# B&R Automation Studio project TD52 (part 145)

#### ECB_Test.st - Implementation code
```iecst
(********************************************************************
 * COPYRIGHT -- INNIO Company
 ********************************************************************
 * Program: ECB_Test
 * File: ECB_Test.st
 * Author: 502423184
 * Created: January 12, 2018
 ********************************************************************
 * Implementation of program ECB_Test
 ********************************************************************)

PROGRAM _INIT

	(** INIT: Disable PBC_Buffer Task *)
	bECB_Buffer_Test	:=	TRUE;

	(** Bit Names **)
	Buffer.Bits[0].used	:=	8;
	Buffer.Bits[1].used	:=	0;
	Buffer.Bits[0].Info[0].Name			:=	'GCB_ON';
	Buffer.Bits[0].Info[1].Name			:=	'Trip_1';
	Buffer.Bits[0].Info[2].Name			:=	'Trip_2';
	Buffer.Bits[0].Info[3].Name			:=	'Trip_3';
	Buffer.Bits[0].Info[4].Name			:=	'GrC_VoltageLow';
	Buffer.Bits[0].Info[5].Name			:=	'GrC_SpeedChange';
	Buffer.Bits[0].Info[6].Name			:=	'GrC_CurrentChange';
	Buffer.Bits[0].Info[7].Name			:=	'FS_IPOffs_Trip';
	Buffer.Bits[1].Info[0].Name			:=	'';
	Buffer.Bits[1].Info[1].Name			:=	'';
	Buffer.Bits[1].Info[2].Name			:=	'';
	Buffer.Bits[1].Info[3].Name			:=	'';

	(** Bit Pattern Names **)
	Buffer.pattern[0].Name		:=	 'PBCNegVoltCheck_';
	Buffer.pattern[1].Name		:=	 'PBCNegPresCheck_';
	Buffer.pattern[2].Name		:=	 'PBCPresSlopeCheck_';
	Buffer.pattern[3].Name		:=	 'PBCSlowDriftCheck_';
	Buffer.pattern[4].Name		:=	 'PBCMemBurst_';
	Buffer.pattern[5].Name		:=	 'PBCSensError_';
	Buffer.pattern[6].Name		:=	 'GlowIgn_';
	Buffer.pattern[7].Name		:=	 'Misfire_I_';
	Buffer.pattern[8].Name		:=	 'Misfire_II_';
	Buffer.pattern[9].Name		:=	 'SkipFire_';
	Buffer.pattern[10].Name		:=	 'LimpHome_';
	Buffer.pattern[11].Name		:=	 'LimpHomeExt_';
	Buffer.pattern[12].Name		:=	 '';
	Buffer.pattern[13].Name		:=	 '';
	Buffer.pattern[14].Name		:=	 '';
	Buffer.pattern[15].Name		:=	 '';
	Buffer.pattern[16].Name		:=	 '';

	Buffer.iCnt_pattern			:=	15;

	(** ui16 Names, Conversions, Signs and Units *)
	iCnt	:=	0;
	FOR iSet:=0 TO 304 BY 16 DO
		Buffer.ui16[iSet].Name 	:=	'Ign_Timing_';		Buffer.ui16[iSet].Co := 100;	Buffer.ui16[iSet].Signed := 1;	Buffer.ui16[iSet].Unit := '°CA';
		iCnt := iCnt +1;	itoa(iCnt,ADR(strCnt));		strcat(ADR(Buffer.ui16[iSet].Name), ADR(strCnt));
	END_FOR
	iCnt	:=	0;
	FOR iSet:=1 TO 305 BY 16 DO
		Buffer.ui16[iSet].Name := 'Knck_Intgr_';		Buffer.ui16[iSet].Co := 10;		Buffer.ui16[iSet].Signed := 1;	Buffer.ui16[iSet].Unit := '%';
		iCnt := iCnt +1;	itoa(iCnt,ADR(strCnt));		strcat(ADR(Buffer.ui16[iSet].Name), ADR(strCnt));
	END_FOR
	iCnt	:=	0;
	FOR iSet:=2 TO 306 BY 16 DO
		Buffer.ui16[iSet].Name := 'U_Ign_';				Buffer.ui16[iSet].Co := 1;		Buffer.ui16[iSet].Signed := 0;	Buffer.ui16[iSet].Unit := 'kV';
		iCnt := iCnt +1;	itoa(iCnt,ADR(strCnt));		strcat(ADR(Buffer.ui16[iSet].Name), ADR(strCnt));
	END_FOR
	iCnt	:=	0;
	FOR iSet:=3 TO 307 BY 16 DO
		Buffer.ui16[iSet].Name := 'PI_Duration_';		Buffer.ui16[iSet].Co := 100;	Buffer.ui16[iSet].Signed := 0;	Buffer.ui16[iSet].Unit := '°CA';
		iCnt := iCnt +1;	itoa(iCnt,ADR(strCnt));		strcat(ADR(Buffer.ui16[iSet].Name), ADR(strCnt));
	END_FOR
	iCnt	:=	0;
	FOR iSet:=4 TO 308 BY 16 DO
		Buffer.ui16[iSet].Name := 'PI_Dur_Map_Offs_';	Buffer.ui16[iSet].Co := 1000;	Buffer.ui16[iSet].Signed := 1;	Buffer.ui16[iSet].Unit := '%';
		iCnt := iCnt +1;	itoa(iCnt,ADR(strCnt));		strcat(ADR(Buffer.ui16[iSet].Name), ADR(strCnt));
	END_FOR
	iCnt	:=	0;
	FOR iSet:=6 TO 310 BY 16 DO
		Buffer.ui16[iSet].Name := 'Pr_Knock_';			Buffer.ui16[iSet].Co := 100;	Buffer.ui16[iSet].Signed := 0;	Buffer.ui16[iSet].Unit := 'bar';
		iCnt := iCnt +1;	itoa(iCnt,ADR(strCnt));		strcat(ADR(Buffer.ui16[iSet].Name), ADR(strCnt));
	END_FOR
	iCnt	:=	0;
	FOR iSet:=7 TO 311 BY 16 DO
		Buffer.ui16[iSet].Name := 'Pr_Knock_Filt_';		Buffer.ui16[iSet].Co := 100;	Buffer.ui16[iSet].Signed := 0;	Buffer.ui16[iSet].Unit := 'bar';
		iCnt := iCnt +1;	itoa(iCnt,ADR(strCnt));		strcat(ADR(Buffer.ui16[iSet].Name), ADR(strCnt));
	END_FOR
	iCnt	:=	0;
	FOR iSet:=8 TO 312 BY 16 DO
		Buffer.ui16[iSet].Name := 'Pr_Peak_';			Buffer.ui16[iSet].Co := 100;	Buffer.ui16[iSet].Signed := 0;	Buffer.ui16[iSet].Unit := 'bar';
		iCnt := iCnt +1;	itoa(iCnt,ADR(strCnt));		strcat(ADR(Buffer.ui16[iSet].Name), ADR(strCnt));
	END_FOR
	iCnt	:=	0;
	FOR iSet:=9 TO 313 BY 16 DO
		Buffer.ui16[iSet].Name := 'Pr_Peak_Filt_';		Buffer.ui16[iSet].Co := 100;	Buffer.ui16[iSet].Signed := 0;	Buffer.ui16[iSet].Unit := 'bar';
		iCnt := iCnt +1;	itoa(iCnt,ADR(strCnt));		strcat(ADR(Buffer.ui16[iSet].Name), ADR(strCnt));
	END_FOR
	iCnt	:=	0;
	FOR iSet:=10 TO 314 BY 16 DO
		Buffer.ui16[iSet].Name := 'Pr_IMEP_';			Buffer.ui16[iSet].Co := 100;	Buffer.ui16[iSet].Signed := 0;	Buffer.ui16[iSet].Unit := 'bar';
		iCnt := iCnt +1;	itoa(iCnt,ADR(strCnt));		strcat(ADR(Buffer.ui16[iSet].Name), ADR(strCnt));
	END_FOR
	iCnt	:=	0;
	FOR iSet:=11 TO 315 BY 16 DO
		Buffer.ui16[iSet].Name := 'Pr_49bfTDC_';		Buffer.ui16[iSet].Co := 100;	Buffer.ui16[iSet].Signed := 0;	Buffer.ui16[iSet].Unit := 'bar';
		iCnt := iCnt +1;	itoa(iCnt,ADR(strCnt));		strcat(ADR(Buffer.ui16[iSet].Name), ADR(strCnt));
	END_FOR
	iCnt	:=	0;
	FOR iSet:=12 TO 316 BY 16 DO
		Buffer.ui16[iSet].Name := 'Pr_49afTDC_';		Buffer.ui16[iSet].Co := 100;	Buffer.ui16[iSet].Signed := 0;	Buffer.ui16[iSet].Unit := 'bar';
		iCnt := iCnt +1;	itoa(iCnt,ADR(strCnt));		strcat(ADR(Buffer.ui16[iSet].Name), ADR(strCnt));
	END_FOR
	iCnt	:=	0;
	FOR iSet:=13 TO 317 BY 16 DO
		Buffer.ui16[iSet].Name := 'MFBvar_';			Buffer.ui16[iSet].Co := 100;	Buffer.ui16[iSet].Signed := 1;	Buffer.ui16[iSet].Unit := '°CA';
		iCnt := iCnt +1;	itoa(iCnt,ADR(strCnt));		strcat(ADR(Buffer.ui16[iSet].Name), ADR(strCnt));
	END_FOR
	iCnt	:=	0;
	FOR iSet:=14 TO 318 BY 16 DO
		Buffer.ui16[iSet].Name := 'Pr_Knock_Lim_';		Buffer.ui16[iSet].Co := 100;	Buffer.ui16[iSet].Signed := 0;	Buffer.ui16[iSet].Unit := 'bar';
		iCnt := iCnt +1;	itoa(iCnt,ADR(strCnt));		strcat(ADR(Buffer.ui16[iSet].Name), ADR(strCnt));
	END_FOR

	Buffer.iCnt_ui16			:=	326;

	(** ui16_H Names, Conversions, Signs and Units *)
	Buffer.ui16_H[0].Name := 'N_Eng';			Buffer.ui16_H[0].Co := 10;		Buffer.ui16_H[0].Signed := 0;	Buffer.ui16_H[0].Unit := 'rpm';
	Buffer.ui16_H[1].Name := 'P_Set';			Buffer.ui16_H[1].Co	:= 1;		Buffer.ui16_H[1].Signed := 0;	Buffer.ui16_H[1].Unit := 'kW';
	Buffer.ui16_H[2].Name := 'P_Act';			Buffer.ui16_H[2].Co := 1;		Buffer.ui16_H[2].Signed	:= 1;	Buffer.ui16_H[2].Unit := 'kW';
	Buffer.ui16_H[3].Name := 'Q_Act';			Buffer.ui16_H[3].Co := 1;		Buffer.ui16_H[3].Signed	:= 1;	Buffer.ui16_H[3].Unit := 'kVAr';
	Buffer.ui16_H[4].Name := 'U_L1L2';			Buffer.ui16_H[4].Co := 1;		Buffer.ui16_H[4].Signed	:= 1;	Buffer.ui16_H[4].Unit := 'V';
	Buffer.ui16_H[5].Name := 'U_L2L3';			Buffer.ui16_H[5].Co := 1;		Buffer.ui16_H[5].Signed	:= 1;	Buffer.ui16_H[5].Unit := 'V';
	Buffer.ui16_H[6].Name := 'U_L3L1';			Buffer.ui16_H[6].Co := 1;		Buffer.ui16_H[6].Signed	:= 1;	Buffer.ui16_H[6].Unit := 'V';
	Buffer.ui16_H[7].Name := 'I_L1';			Buffer.ui16_H[7].Co := 1;		Buffer.ui16_H[7].Signed	:= 1;	Buffer.ui16_H[7].Unit := 'A';
	Buffer.ui16_H[8].Name := 'I_L2';			Buffer.ui16_H[8].Co := 1;		Buffer.ui16_H[8].Signed	:= 1;	Buffer.ui16_H[8].Unit := 'A';
	Buffer.ui16_H[9].Name := 'I_L3';			Buffer.ui16_H[9].Co := 1;		Buffer.ui16_H[9].Signed	:= 1;	Buffer.ui16_H[9].Unit := 'A';
	Buffer.ui16_H[10].Name := 'Frequency';		Buffer.ui16_H[10].Co := 1000;	Buffer.ui16_H[10].Signed := 0;	Buffer.ui16_H[10].Unit := 'Hz';
	Buffer.ui16_H[11].Name := 'CosPhi';			Buffer.ui16_H[11].Co := 100;	Buffer.ui16_H[11].Signed := 1;	Buffer.ui16_H[11].Unit := '';
	Buffer.ui16_H[12].Name := 'Lambda_Set';		Buffer.ui16_H[12].Co := 1000;	Buffer.ui16_H[12].Signed := 0;	Buffer.ui16_H[12].Unit := '';
	Buffer.ui16_H[13].Name := 'Pr_Leanox_Set';	Buffer.ui16_H[13].Co := 1000;	Buffer.ui16_H[13].Signed := 0;	Buffer.ui16_H[13].Unit := '';
	Buffer.ui16_H[14].Name := 'N_TCHP_A';		Buffer.ui16_H[14].Co := 0.1;	Buffer.ui16_H[14].Signed := 0;	Buffer.ui16_H[14].Unit := 'rpm';
	Buffer.ui16_H[15].Name := 'N_TCHP_B';		Buffer.ui16_H[15].Co := 0.1;	Buffer.ui16_H[15].Signed := 0;	Buffer.ui16_H[15].Unit := 'rpm';
	Buffer.ui16_H[16].Name := 'N_TCLP_A';		Buffer.ui16_H[16].Co := 0.1;	Buffer.ui16_H[16].Signed := 0;	Buffer.ui16_H[16].Unit := 'rpm';
	Buffer.ui16_H[17].Name := 'N_TCLP_B';		Buffer.ui16_H[17].Co := 0.1;	Buffer.ui16_H[17].Signed := 0;	Buffer.ui16_H[17].Unit := 'rpm';
	Buffer.ui16_H[18].Name := 'Pr_GR_Act';		Buffer.ui16_H[18].Co := 1000;	Buffer.ui16_H[18].Signed := 0;	Buffer.ui16_H[18].Unit := 'bar';
	Buffer.ui16_H[19].Name := 'Pr_GR_Set';		Buffer.ui16_H[19].Co := 1000;	Buffer.ui16_H[19].Signed := 0;	Buffer.ui16_H[19].Unit := 'bar';
	Buffer.ui16_H[20].Name := 'Pr_PC_Act';		Buffer.ui16_H[20].Co := 1000;	Buffer.ui16_H[20].Signed := 0;	Buffer.ui16_H[20].Unit := 'bar';
	Buffer.ui16_H[21].Name := 'Pr_PC_Set';		Buffer.ui16_H[21].Co := 1000;	Buffer.ui16_H[21].Signed := 0;	Buffer.ui16_H[21].Unit := 'bar';
	Buffer.ui16_H[22].Name := 'Pr_Crank_Case';	Buffer.ui16_H[22].Co := 1000;	Buffer.ui16_H[22].Signed := 1;	Buffer.ui16_H[22].Unit := 'mbar';
	Buffer.ui16_H[23].Name := 'Pos_CBV_Set';	Buffer.ui16_H[23].Co := 1000;	Buffer.ui16_H[23].Signed := 0;	Buffer.ui16_H[23].Unit := '';
	Buffer.ui16_H[24].Name := 'Pos_CBV_Act_A1';	Buffer.ui16_H[24].Co := 1000;	Buffer.ui16_H[24].Signed := 0;	Buffer.ui16_H[24].Unit := '';
	Buffer.ui16_H[25].Name := 'Pos_CBV_Act_B1';	Buffer.ui16_H[25].Co := 1000;	Buffer.ui16_H[25].Signed := 0;	Buffer.ui16_H[25].Unit := '';
	Buffer.ui16_H[26].Name := 'Pos_WG_Set';		Buffer.ui16_H[26].Co := 1000;	Buffer.ui16_H[26].Signed := 0;	Buffer.ui16_H[26].Unit := '';
	Buffer.ui16_H[27].Name := 'Pos_WG_Act_A';	Buffer.ui16_H[27].Co := 1000;	Buffer.ui16_H[27].Signed := 0;	Buffer.ui16_H[27].Unit := '';
	Buffer.ui16_H[28].Name := 'Pos_WG_Act_B';	Buffer.ui16_H[28].Co := 1000;	Buffer.ui16_H[28].Signed := 0;	Buffer.ui16_H[28].Unit := '';
	Buffer.ui16_H[29].Name := 'Pr_P1HP_A';		Buffer.ui16_H[29].Co := 1000;	Buffer.ui16_H[29].Signed := 0;	Buffer.ui16_H[29].Unit := 'bar';
	Buffer.ui16_H[30].Name := 'Pr_P1HP_B';		Buffer.ui16_H[30].Co := 1000;	Buffer.ui16_H[30].Signed := 0;	Buffer.ui16_H[30].Unit := 'bar';
	Buffer.ui16_H[31].Name := 'Pr_P2s_A';		Buffer.ui16_H[31].Co := 1000;	Buffer.ui16_H[31].Signed := 0;	Buffer.ui16_H[31].Unit := 'bar';
	Buffer.ui16_H[32].Name := 'Pr_P2s_B';		Buffer.ui16_H[32].Co := 1000;	Buffer.ui16_H[32].Signed := 0;	Buffer.ui16_H[32].Unit := 'bar';
	Buffer.ui16_H[33].Name := 'Pr_P3HP_A';		Buffer.ui16_H[33].Co := 1000;	Buffer.ui16_H[33].Signed := 0;	Buffer.ui16_H[33].Unit := 'bar';
	Buffer.ui16_H[34].Name := 'Pr_P3HP_B';		Buffer.ui16_H[34].Co := 1000;	Buffer.ui16_H[34].Signed := 0;	Buffer.ui16_H[34].Unit := 'bar';
	Buffer.ui16_H[35].Name := 'Pr_P3LP_A';		Buffer.ui16_H[35].Co := 1000;	Buffer.ui16_H[35].Signed := 0;	Buffer.ui16_H[35].Unit := 'bar';
	Buffer.ui16_H[36].Name := 'Pr_P3LP_B';		Buffer.ui16_H[36].Co := 1000;	Buffer.ui16_H[36].Signed := 0;	Buffer.ui16_H[36].Unit := 'bar';
	Buffer.ui16_H[37].Name := 'Pr_P4LP_A';		Buffer.ui16_H[37].Co := 1000;	Buffer.ui16_H[37].Signed := 0;	Buffer.ui16_H[37].Unit := 'bar';
	Buffer.ui16_H[38].Name := 'Pr_P4LP_B';		Buffer.ui16_H[38].Co := 1000;	Buffer.ui16_H[38].Signed := 0;	Buffer.ui16_H[38].Unit := 'bar';
	Buffer.ui16_H[39].Name := 'Pr_ECW';			Buffer.ui16_H[39].Co := 1000;	Buffer.ui16_H[39].Signed := 0;	Buffer.ui16_H[39].Unit := 'bar';
	Buffer.ui16_H[40].Name := 'Pr_EO';			Buffer.ui16_H[40].Co := 1000;	Buffer.ui16_H[40].Signed := 0;	Buffer.ui16_H[40].Unit := 'bar';
	Buffer.ui16_H[41].Name := 'NOx_Sensor_1';	Buffer.ui16_H[41].Co := 1;		Buffer.ui16_H[41].Signed := 0;	Buffer.ui16_H[41].Unit := '';
	Buffer.ui16_H[42].Name := 'NOx_Sensor_2';	Buffer.ui16_H[42].Co := 1;		Buffer.ui16_H[42].Signed := 0;	Buffer.ui16_H[42].Unit := '';
	Buffer.ui16_H[43].Name := 'O2_Sensor_1';	Buffer.ui16_H[43].Co := 1;		Buffer.ui16_H[43].Signed := 0;	Buffer.ui16_H[43].Unit := '';
	Buffer.ui16_H[44].Name := 'O2_Sensor_2';	Buffer.ui16_H[44].Co := 1;		Buffer.ui16_H[44].Signed := 0;	Buffer.ui16_H[44].Unit := '';
	Buffer.ui16_H[45].Name := '';				Buffer.ui16_H[45].Co := 0;		Buffer.ui16_H[45].Signed := 0;	Buffer.ui16_H[45].Unit := '';
	Buffer.ui16_H[46].Name := '';				Buffer.ui16_H[46].Co := 0;		Buffer.ui16_H[46].Signed := 0;	Buffer.ui16_H[46].Unit := '';

	Buffer.iCnt_ui16_H	:=	44;

	(** ui16_L Names, Conversions, Signs and Units *)
	FOR iSet:=0 TO 56 DO
		Buffer.ui16_low[iSet].Signed	:= 0;
		Buffer.ui16_low[iSet].Unit		:= '°C';
		Buffer.ui16_low[iSet].Co		:=	100;
	END_FOR

	Buffer.ui16_low[0].Name := 'T_T2s';
	Buffer.ui16_low[1].Name := 'T_T3HP_A';		Buffer.ui16_low[1].Co := 10;	(* nur EG temps mit Conversion 10 *)
	Buffer.ui16_low[2].Name := 'T_T3HP_B';		Buffer.ui16_low[2].Co := 10;
	Buffer.ui16_low[3].Name := 'T_T3LP_A';		Buffer.ui16_low[3].Co := 10;
	Buffer.ui16_low[4].Name := 'T_T3LP_B';		Buffer.ui16_low[4].Co := 10;
	Buffer.ui16_low[5].Name := 'T_EG_LimMax';	Buffer.ui16_low[5].Co := 10;

	iCnt	:=	0; (* zyl 1 bis 11 *)
	FOR iSet:=6 TO 36 BY 3 DO
		iCnt := iCnt +1;	itoa(iCnt,ADR(strCnt));
		Buffer.ui16_low[iSet].Name		:= 'T_EG_Cyl_';		strcat(ADR(Buffer.ui16_low[iSet].Name), ADR(strCnt));
		Buffer.ui16_low[iSet+1].Name	:= 'T_CBearing_';	strcat(ADR(Buffer.ui16_low[iSet+1].Name), ADR(strCnt));
		Buffer.ui16_low[iSet+2].Name	:= 'T_MBearing_';	strcat(ADR(Buffer.ui16_low[iSet+2].Name), ADR(strCnt));
	END_FOR
	iCnt	:=	11;	(* zyl 12 bis 20 *)
	FOR iSet:=39 TO 55 BY 2 DO
		iCnt := iCnt +1;	itoa(iCnt,ADR(strCnt));
		Buffer.ui16_low[iSet].Name		:= 'T_EG_Cyl_';		strcat(ADR(Buffer.ui16_low[iSet].Name), ADR(strCnt));
		Buffer.ui16_low[iSet+1].Name	:= 'T_CBearing_';	strcat(ADR(Buffer.ui16_low[iSet+1].Name), ADR(strCnt));
	END_FOR

	Buffer.ui16_low[57].Name := '';	Buffer.ui16_low[57].Co := 0;	Buffer.ui16_low[57].Signed := 0;	Buffer.ui16_low[57].Unit := '';

	Buffer.iCnt_ui16_low		:=	56;

END_PROGRAM

PROGRAM _CYCLIC

(** 1: is PBCMem enabled? *)
IF bPBC_Mem_Ena THEN

(** 6: save data to buffer? @control *)
	IF 	bPBC_NewData AND bPBC_Record THEN

(** 6.1: save the time *)
		Buffer.timer[iCnt_Cycle]	:= tiStamp;
(* _______________________________________________________ FAKE BITS _______________________________________________________ *)

		Buffer.Bits[0].ucData[iCnt_Cycle]	:=	1;
		Buffer.Bits[1].ucData[iCnt_Cycle]	:=	0;
		FOR iSet:= 1 TO 16 DO
			Buffer.pattern[iSet].BitPattern[iCnt_Cycle]	:=	INT_TO_UDINT(iCnt_Cycle) + INT_TO_UDINT(iCnt_Cycle)*1000;
		END_FOR

(* _______________________________________________________ FAKE PATTERNS _______________________________________________________ *)

	iCnt_Cycle10	:=	LIMIT(0,iCnt_Cycle/10,100);

	iCnt := 0;	FOR iSet:=0 TO 304 BY 16 DO			Buffer.ui16[iSet].Data[iCnt_Cycle] := 1914;			END_FOR
	iCnt := 0;	FOR iSet:=1 TO 305 BY 16 DO			Buffer.ui16[iSet].Data[iCnt_Cycle] := 43;			END_FOR
	iCnt := 0;	FOR iSet:=2 TO 306 BY 16 DO			Buffer.ui16[iSet].Data[iCnt_Cycle] := 15;			END_FOR
	iCnt := 0;	FOR iSet:=3 TO 307 BY 16 DO			Buffer.ui16[iSet].Data[iCnt_Cycle] := 6210;			END_FOR
	iCnt := 0;	FOR iSet:=4 TO 308 BY 16 DO			Buffer.ui16[iSet].Data[iCnt_Cycle] := 1492;			END_FOR
(* 5 fehlt *)
	iCnt := 0;	FOR iSet:=6 TO 310 BY 16 DO			Buffer.ui16[iSet].Data[iCnt_Cycle] := 166;			END_FOR
	iCnt := 0;	FOR iSet:=7 TO 311 BY 16 DO			Buffer.ui16[iSet].Data[iCnt_Cycle] := 166;			END_FOR
	iCnt := 0;	FOR iSet:=8 TO 312 BY 16 DO			Buffer.ui16[iSet].Data[iCnt_Cycle] := 15816;		END_FOR
	iCnt := 0;	FOR iSet:=9 TO 313 BY 16 DO			Buffer.ui16[iSet].Data[iCnt_Cycle] := 15816;		END_FOR
	iCnt := 0;	FOR iSet:=10 TO 314 BY 16 DO		Buffer.ui16[iSet].Data[iCnt_Cycle] := 2611;			END_FOR
	iCnt := 0;	FOR iSet:=11 TO 315 BY 16 DO		Buffer.ui16[iSet].Data[iCnt_Cycle] := 2233;			END_FOR
	iCnt := 0;	FOR iSet:=12 TO 316 BY 16 DO		Buffer.ui16[iSet].Data[iCnt_Cycle] := 5914;			END_FOR
	iCnt := 0;	FOR iSet:=13 TO 317 BY 16 DO		Buffer.ui16[iSet].Data[iCnt_Cycle] := 1000;			END_FOR
	iCnt := 0;	FOR iSet:=14 TO 318 BY 16 DO		Buffer.ui16[iSet].Data[iCnt_Cycle] := 2233;			END_FOR
	iCnt := 0;	FOR iSet:=15 TO 319 BY 16 DO		Buffer.ui16[iSet].Data[iCnt_Cycle] := 65293;		END_FOR
	iCnt := 0;	FOR iSet:=16 TO 320 BY 16 DO		Buffer.ui16[iSet].Data[iCnt_Cycle] := 166;			END_FOR

	Buffer.ui16_H[0].Hi[iCnt_Cycle] := 10000;		Buffer.ui16_H[0].Lo[iCnt_Cycle] := 9990;
	Buffer.ui16_H[1].Hi[iCnt_Cycle] := 10380;		Buffer.ui16_H[1].Lo[iCnt_Cycle] := 10340;
	Buffer.ui16_H[2].Hi[iCnt_Cycle] := 10434;		Buffer.ui16_H[2].Lo[iCnt_Cycle] := 10428;
	Buffer.ui16_H[3].Hi[iCnt_Cycle] := 26;			Buffer.ui16_H[3].Lo[iCnt_Cycle] := 34;
	Buffer.ui16_H[4].Hi[iCnt_Cycle] := 10621;		Buffer.ui16_H[4].Lo[iCnt_Cycle] := 10622;
	Buffer.ui16_H[5].Hi[iCnt_Cycle] := 10621;		Buffer.ui16_H[5].Lo[iCnt_Cycle] := 10622;
	Buffer.ui16_H[6].Hi[iCnt_Cycle] := 10621;		Buffer.ui16_H[6].Lo[iCnt_Cycle] := 10622;
	Buffer.ui16_H[7].Hi[iCnt_Cycle] := 568;			Buffer.ui16_H[7].Lo[iCnt_Cycle] := 569;
	Buffer.ui16_H[8].Hi[iCnt_Cycle] := 568;			Buffer.ui16_H[8].Lo[iCnt_Cycle] := 568;
	Buffer.ui16_H[9].Hi[iCnt_Cycle] := 574;			Buffer.ui16_H[9].Lo[iCnt_Cycle] := 571;
	Buffer.ui16_H[10].Hi[iCnt_Cycle] := 50000;		Buffer.ui16_H[10].Lo[iCnt_Cycle] := 49990;
	Buffer.ui16_H[11].Hi[iCnt_Cycle] := 100;		Buffer.ui16_H[11].Lo[iCnt_Cycle] := 100;
	Buffer.ui16_H[12].Hi[iCnt_Cycle] := 1973;		Buffer.ui16_H[12].Lo[iCnt_Cycle] := 1973;
	Buffer.ui16_H[13].Hi[iCnt_Cycle] := 7630;		Buffer.ui16_H[13].Lo[iCnt_Cycle] := 7630;
	Buffer.ui16_H[14].Hi[iCnt_Cycle] := 2760;		Buffer.ui16_H[14].Lo[iCnt_Cycle] := 2763;
	Buffer.ui16_H[15].Hi[iCnt_Cycle] := 2753;		Buffer.ui16_H[15].Lo[iCnt_Cycle] := 2753;
	Buffer.ui16_H[16].Hi[iCnt_Cycle] := 2625;		Buffer.ui16_H[16].Lo[iCnt_Cycle] := 2596;
	Buffer.ui16_H[17].Hi[iCnt_Cycle] := 2594;		Buffer.ui16_H[17].Lo[iCnt_Cycle] := 2594;
	Buffer.ui16_H[18].Hi[iCnt_Cycle] := 8815;		Buffer.ui16_H[18].Lo[iCnt_Cycle] := 8818;
	Buffer.ui16_H[19].Hi[iCnt_Cycle] := 8853;		Buffer.ui16_H[19].Lo[iCnt_Cycle] := 8853;
	Buffer.ui16_H[20].Hi[iCnt_Cycle] := 5369;		Buffer.ui16_H[20].Lo[iCnt_Cycle] := 5369;
	Buffer.ui16_H[21].Hi[iCnt_Cycle] := 6851;		Buffer.ui16_H[21].Lo[iCnt_Cycle] := 6851;
	Buffer.ui16_H[22].Hi[iCnt_Cycle] := 62867;		Buffer.ui16_H[22].Lo[iCnt_Cycle] := 62987;
	Buffer.ui16_H[23].Hi[iCnt_Cycle] := 28;			Buffer.ui16_H[23].Lo[iCnt_Cycle] := 28;
	Buffer.ui16_H[24].Hi[iCnt_Cycle] := 29;			Buffer.ui16_H[24].Lo[iCnt_Cycle] := 28;
	Buffer.ui16_H[25].Hi[iCnt_Cycle] := 26;			Buffer.ui16_H[25].Lo[iCnt_Cycle] := 25;
	Buffer.ui16_H[26].Hi[iCnt_Cycle] := 478;		Buffer.ui16_H[26].Lo[iCnt_Cycle] := 478;
	Buffer.ui16_H[27].Hi[iCnt_Cycle] := 487;		Buffer.ui16_H[27].Lo[iCnt_Cycle] := 486;
	Buffer.ui16_H[28].Hi[iCnt_Cycle] := 488;		Buffer.ui16_H[28].Lo[iCnt_Cycle] := 488;
	Buffer.ui16_H[29].Hi[iCnt_Cycle] := 3210;		Buffer.ui16_H[29].Lo[iCnt_Cycle] := 3213;
	Buffer.ui16_H[30].Hi[iCnt_Cycle] := 3236;		Buffer.ui16_H[30].Lo[iCnt_Cycle] := 3233;
	Buffer.ui16_H[31].Hi[iCnt_Cycle] := 6732;		Buffer.ui16_H[31].Lo[iCnt_Cycle] := 6733;
	Buffer.ui16_H[32].Hi[iCnt_Cycle] := 6662;		Buffer.ui16_H[32].Lo[iCnt_Cycle] := 6662;
	Buffer.ui16_H[33].Hi[iCnt_Cycle] := 4605;		Buffer.ui16_H[33].Lo[iCnt_Cycle] := 4621;
	Buffer.ui16_H[34].Hi[iCnt_Cycle] := 4675;		Buffer.ui16_H[34].Lo[iCnt_Cycle] := 4675;
	Buffer.ui16_H[35].Hi[iCnt_Cycle] := 2864;		Buffer.ui16_H[35].Lo[iCnt_Cycle] := 2873;
	Buffer.ui16_H[36].Hi[iCnt_Cycle] := 2879;		Buffer.ui16_H[36].Lo[iCnt_Cycle] := 2870;
	Buffer.ui16_H[37].Hi[iCnt_Cycle] := 1026;		Buffer.ui16_H[37].Lo[iCnt_Cycle] := 1029;
	Buffer.ui16_H[38].Hi[iCnt_Cycle] := 1021;		Buffer.ui16_H[38].Lo[iCnt_Cycle] := 1017;
	Buffer.ui16_H[39].Hi[iCnt_Cycle] := 2147;		Buffer.ui16_H[39].Lo[iCnt_Cycle] := 2128;
	Buffer.ui16_H[40].Hi[iCnt_Cycle] := 5797;		Buffer.ui16_H[40].Lo[iCnt_Cycle] := 5794;
	Buffer.ui16_H[41].Hi[iCnt_Cycle] := 216;		Buffer.ui16_H[41].Lo[iCnt_Cycle] := 216;
	Buffer.ui16_H[42].Hi[iCnt_Cycle] := 219;		Buffer.ui16_H[42].Lo[iCnt_Cycle] := 219;
	Buffer.ui16_H[43].Hi[iCnt_Cycle] := 0;			Buffer.ui16_H[43].Lo[iCnt_Cycle] := 0;
	Buffer.ui16_H[44].Hi[iCnt_Cycle] := 0;			Buffer.ui16_H[44].Lo[iCnt_Cycle] := 0;
	Buffer.ui16_H[45].Hi[iCnt_Cycle] := 0;			Buffer.ui16_H[45].Lo[iCnt_Cycle] := 0;
	Buffer.ui16_H[46].Hi[iCnt_Cycle] := 0;			Buffer.ui16_H[46].Lo[iCnt_Cycle] := 0;

	Buffer.ui16_low[0].Data[iCnt_Cycle10] := 7545;
	Buffer.ui16_low[1].Data[iCnt_Cycle10] := 5366;
	Buffer.ui16_low[2].Data[iCnt_Cycle10] := 5366;
	Buffer.ui16_low[3].Data[iCnt_Cycle10] := 4577;
	Buffer.ui16_low[4].Data[iCnt_Cycle10] := 4605;
	Buffer.ui16_low[5].Data[iCnt_Cycle10] := 6000;

	FOR iSet:=6 TO 36 BY 3 DO
		Buffer.ui16_low[iSet].Data[iCnt_Cycle10]	:= 52900;		(* 6,9,12 bis 36 *)
		Buffer.ui16_low[iSet+1].Data[iCnt_Cycle10]	:= 10100;		(* 7,10,13 bis 37 *)
		Buffer.ui16_low[iSet+2].Data[iCnt_Cycle10]	:= 10120;		(* 8,11,14 bis 38 *)
	END_FOR
	FOR iSet:=39 TO 55 BY 2 DO
		Buffer.ui16_low[iSet].Data[iCnt_Cycle10]	:= 52900;		(* 39,41,43 bis 55 *)
		Buffer.ui16_low[iSet+1].Data[iCnt_Cycle10]	:= 10100;		(* 40,42,44 bis 56 *)
	END_FOR

	Buffer.ui16_low[57].Data[iCnt_Cycle10] := 0;

(* ________________________________________________________________________ TEST ____________________________________ *)

		bPBC_NewData	:=	FALSE;

(** 6.6: increase cycle counter *)
		iCnt_Cycle := (iCnt_Cycle +1) MOD iBufferSize;
	END_IF

	bWarn_Buffer	:=	iTC_Max = INT_TO_UINT(Buffer.iCnt_ui16_H) OR
						iEC_Max = INT_TO_UINT(Buffer.iCnt_ui16) OR
						iSC_Max = INT_TO_UINT(Buffer.iCnt_ui16_low) OR
						iPC_Max = INT_TO_UINT(Buffer.iCnt_pattern);

END_IF

END_PROGRAM

PROGRAM _EXIT

	(** EXIT: Enable PBC_Buffer Task *)
	bECB_Buffer_Test	:=	FALSE;

END_PROGRAM
```

#### ECB_Test.var - Local variables
```iecst
(********************************************************************
 * COPYRIGHT -- INNIO Company
 ********************************************************************
 * Program: ECB_Test
 * File: ECB_Test.var
 * Author: 502423184
 * Created: January 12, 2018
 ********************************************************************
 * Local variables of program ECB_Test
 ********************************************************************)
VAR
	iCnt : DINT := 0;
	strCnt : STRING[5];
	iSet : DINT;
	iCnt_Cycle10 : INT;
END_VAR
```

### Program Logical/CBM/PBCMemV2/PBC_Obj (IEC) - Save Object

#### PBC_Obj.st - Cyclic code
```iecst
(*******************************************************************************
AGGR: read and write DIA.NE XT parameter to flash memory	(cyclic)

This code is confidential and proprietary to the INNIO Company.
It may not be used in any form, or reproduced in any manner, without the express
written permission of the INNIO Company.
Copyright, INNIO Company, 2019

Customized modifications: -
------------------------

History:
-------
V3.50.3		05-11-2014	Caks,		generated
			18-11-2014	Caks,		added File-Read Check
			03-12-2014	Caks,		added: Rod and Main bearing temperature
			05-12-2014	Caks,		added: Time to Structure and File
V3.50.4		12-12-2014	Perktold,	set bWrite to FALSE in case of byStep = 7
			17-12-2014	Perktod, 	Bugfix Timestamp
V3.50.5		08-01-2015	Perktold,	Aenderung Dateinamen
			09-02-2015	Perktold,	Z636 - "+13"
V4.02.0		09-03-2015	Caks,		ported to XT4
V4.04.0		28-06-2016	502423184	added EXIT routine
V4.05.0		28-09-2016	502423184	new Version, created from old file
V4.06.0		30-10-2017	502423184	added all changes from spec, also added improved(faster and secure) strcat function
			29-01-2018	502423184	bugfix of time and slow cycle data regarding not filled buffer
			24-04-2018	502423184	new easy way setting up triggers in one line
V4.06.1		16-11-2018	502423184	release version, removed clock_ms()
V4.07.0		21-03-2019	Waldhart	footer increased
			29-03-2023	Kafka,		CBM HMI Handshake for ECBMem Files

Instructions for use:
--------------------

100ms Task class

Outstandings:
------------
*******************************************************************************)

PROGRAM _INIT

(** A: Version *)
	strVersion			:=	'4.14.00';

(** B: Initialize variables *)
	bECB_Lock		:=	FALSE;
	aT				:=	ADR(szTemp);
	aData			:=	ADR(szData);
	iStep 			:=	_IDLE;

	strcpy(ADR(ModulName),ADR('CBM::PBCMem'));

	pm_len			:=	SIZEOF(DerString);	(* define data length of permenent memory  		*)

	DatObjInfo_01.enable		:=	TRUE;
	DatObjInfo_01.pName			:=	ADR(ModulName);

	DatObjCreate_01.enable		:=	TRUE;			(* enable create permanent memory data module FUB 		*)
	DatObjCreate_01.grp			:=	0;				(* must to be set to zero                  				*)
	DatObjCreate_01.pName		:=	ADR(ModulName);	(* set permanent memory data module name             	*)
	DatObjCreate_01.len			:=	pm_len;			(* set length of permanent memory data module         	*)
	DatObjCreate_01.MemType		:=	doUSRROM;		(* create permanent memory data module at USERROM   	*)
	DatObjCreate_01.Option		:=	0;				(* cyclic checksum monitoring is on            			*)
	DatObjCreate_01.pCpyData	:=	0;				(* no data will be copied do the perm. mem. data module	*)

	DatObjWrite_01.enable		:=	TRUE;			(* enable permanent memory data module read FUB 		*)
	DatObjWrite_01.Offset		:=	0;				(* start at memory offest zero                  		*)
	DatObjWrite_01.pSource		:=	ADR(DerString);	(* set permanent memory data module name            	*)
	DatObjWrite_01.len			:=	pm_len;			(* set length ofpermanent memory data module        	*)

(** C: Functionality test and validation *)
	TON_15min.PT 	:= T#15m;
	bTest_Ena		:=	FALSE;

(** D: ATD extension *)
	iLogicSize_1	:=	MAX(0,UDINT_TO_INT(SIZEOF(logicMatrix_1) / MAX(1, SIZEOF(logicMatrix_1[0]))) - 1);
	iLogicSize_2	:=	MAX(0,UDINT_TO_INT(SIZEOF(logicMatrix_2) / MAX(1, SIZEOF(logicMatrix_2[0]))) - 1);

END_PROGRAM

PROGRAM _CYCLIC

(** 1: Test and Validation *)
	IF bTest_Ena THEN
		TON_15min.IN := NOT TON_15min.Q;
		TON_15min();

		IF TON_15min.Q THEN
			iStep := _BEGIN;
		END_IF
	END_IF

(** 2: if recording of the buffer is done then initialiate file write *)
	IF EDGENEG(bPBC_Record) AND bPBC_Write AND bPBC_Mem_Ena THEN
		iStep 		:=	_BEGIN;
		bWrite		:=	TRUE;
	END_IF

(** 3: when write process is done then reset event bit *)
	IF EDGENEG(bWrite) THEN
		bPBC_Write		:=	FALSE;
	END_IF

(** 4: State Machine *)
	CASE iStep OF
(** 4.1: create filename *)
	_BEGIN:
		strFile			:=	'';																				(* Set Filename *)
		WRITE_Date(ADR(strFile),tRealTime);																		(* Date *)
		strcat(ADR(strFile), ADR('_ECB'));																		(* _Name *)
		strcat(ADR(strFile), ADR('_'));	strcat(ADR(strFile), ADR(IN_CB.szOrderID));								(* _OrderID *)
		strcat(ADR(strFile), ADR('_'));	itoa(IN_CB.iEngID, 	 ADR(strTemp));	strcat(ADR(strFile), ADR(strTemp));	(* _EngineID *)
		strcat(ADR(strFile), ADR('_'));	strcat(ADR(strFile), ADR(Buffer.TrigMode[iPBC_Trigger].Name));			(* _Mode *)
		strcat(ADR(strFile), ADR('.csv'));																		(* .csv *)
		iStep		:=	_HEAD;
(** 4.1: create specific header *)
	_HEAD:
		szHeader		:=	'';
		aH				:=	ADR(szHeader);
		FOR iCnt:=0 TO Buffer.iCnt_HS DO																	(* StringData 		*)
			strcat(aH,ADR(Buffer.HeaderS[iCnt].Name));		strcat(aH,ADR(';'));								(* Name;		*)
			strcat(aH,ADR(Buffer.HeaderS[iCnt].Value));		strcat(aH,ADR(';$n'));								(* Value; Return*)
		END_FOR
		FOR iCnt:=0 TO Buffer.iCnt_H12 DO																	(* Array Data 12 	*)
			strcat(aH,ADR(Buffer.Header12[iCnt].Name));		strcat(aH,ADR(';'));								(* Name;		*)
			strcat(aH,ADR(Buffer.Header12[iCnt].Unit));		strcat(aH,ADR(';'));								(* Unit;		*)
			FOR i:= 1 TO xEngType.NumberOfCylinder/2 DO
				WRITE_REAL(Buffer.Header12[iCnt].Value[i], Buffer.Header12[iCnt].Co, aH);						(* Value;		*)
			END_FOR
			strcat(aH,ADR('$n'));																				(* Return		*)
		END_FOR
		FOR iCnt:=0 TO Buffer.iCnt_H DO																		(* standart data 	*)
			strcat(aH,ADR(Buffer.Header[iCnt].Name));		strcat(aH,ADR(';'));								(* Name;		*)
			WRITE_REAL(Buffer.Header[iCnt].Value, Buffer.Header[iCnt].Co, aH);									(* Value;		*)
			strcat(aH,ADR(Buffer.Header[iCnt].Unit));		strcat(aH,ADR(';$n'));								(* Unit; Return	*)
		END_FOR
		strcat(aH, ADR(strLine));																			(* ------------ *)
		iStep		:=	_HEAD1;
(** 4.2: create header for continous data *)
	_HEAD1,_HEAD2:
		bName	:=	iStep = _HEAD1;																			(* Name / Unit		*)
		IF bName THEN		strcat(aH,ADR('Time;'));															(* Time;		*)
		ELSE				strcat(aH,ADR('s;'));																(* s;			*)
		END_IF
		FOR iCnt_B:=0 TO iBits_Max DO																		(* single bits 		*)
			FOR iCnt:=0 TO USINT_TO_INT(Buffer.Bits[iCnt_B].used)-1 DO
				IF bName THEN	strcat(aH,ADR(Buffer.Bits[iCnt_B].Info[iCnt].Name));	END_IF					(* Name			*)
				strcat(aH,ADR(';'));																			(* ;			*)
			END_FOR
		END_FOR
		IF Buffer.iCnt_pattern > 0 THEN
			FOR iCnt:=0 TO Buffer.iCnt_pattern DO																(* bit patterns 	*)
				FOR iCyl:=1 TO xEngType.NumberOfCylinder DO
					IF bName THEN strcat(aH,ADR(Buffer.pattern[iCnt].Name)); itoa(iCyl,aT); strcat(aH,aT); END_IF	(* Name_Cyl		*)
					strcat(aH,ADR(';'));																			(* ;			*)
				END_FOR
			END_FOR
		END_IF
		FOR iCnt:=0 TO Buffer.iCnt_ui16_H DO																(* task cycle data 	*)
			IF bName THEN	strcat(aH,ADR(Buffer.ui16_H[iCnt].Name));	strcat(aH,ADR('_Min;'));				(* Name_Min;	*)
							strcat(aH,ADR(Buffer.ui16_H[iCnt].Name));	strcat(aH,ADR('_Max;'));				(* Name_Max;	*)
			ELSE			strcat(aH,ADR(Buffer.ui16_H[iCnt].Unit));	strcat(aH,ADR(';'));					(* Unit;		*)
							strcat(aH,ADR(Buffer.ui16_H[iCnt].Unit));	strcat(aH,ADR(';'));					(* Unit;		*)
			END_IF
		END_FOR
		FOR iCnt:=0 TO Buffer.iCnt_ui16 DO																	(* engine cycle data *)
			IF bName THEN	strcat(aH,ADR(Buffer.ui16[iCnt].Name));		strcat(aH,ADR(';'));					(* Name;		*)
			ELSE			strcat(aH,ADR(Buffer.ui16[iCnt].Unit));		strcat(aH,ADR(';'));					(* Unit;		*)
			END_IF
		END_FOR
		FOR iCnt:=0 TO Buffer.iCnt_ui16_low DO																(* slow changing data *)
			IF bName THEN	strcat(aH,ADR(Buffer.ui16_low[iCnt].Name));	strcat(aH,ADR(';'));					(* Name;		*)
			ELSE			strcat(aH,ADR(Buffer.ui16_low[iCnt].Unit));	strcat(aH,ADR(';'));					(* Unit;		*)
			END_IF
		END_FOR
		strcat(aH,ADR('$n'));																				(* Return		*)
		IF bName THEN		iStep	:=	_HEAD2;																(* next Line Units *)
		ELSE				iStep	:=	_LOCK;																(* next step *)
		END_IF
(** 4.3: waiting for TCBMem if in write process *)
	_LOCK:
		IF NOT bTCB_Lock THEN
			iStep		:=	_STR;
			bECB_Lock	:=	TRUE;
		END_IF
(** 4.4: fill data string with header *)
	_STR:
		szData		:=	'';
		strcat(aData, ADR('<PBC_NAME>'));																						(* ------------ *)
		strcat(aData, ADR(strFile));																							(* file name *)
		strcat(aData, ADR('</PBC_NAME><PBC_FILE>'));																			(* ------------ *)
		strcat(aData, ADR(strGEProp));																							(* GE prop info *)
		strcat(aData, ADR(strLine));																							(* ------------ *)
		strcat(aData, ADR('File_Version;'));	WRITE_STRING(ADR(strVersion),aData);				strcat(aData, ADR('$n'));	(* File version *)
		strcat(aData, ADR('Creation_Date;'));	WRITE_TS(tTimeStamp, aData);						strcat(aData, ADR('$n'));	(* Date & Time *)
		strcat(aData, ADR('J_Number;'));		WRITE_STRING(ADR(IN_CB.szOrderID),aData);			strcat(aData, ADR('$n'));	(* J Number *)
		strcat(aData, ADR('Motor_Number;'));	WRITE_DINT(IN_CB.iEngID,aData);						strcat(aData, ADR('$n'));	(* Serial ID *)
		strcat(aData, ADR('Engine_Type;'));		WRITE_DINT(xEngType.Motortype,aData);				strcat(aData, ADR('$n'));	(* Engine Type *)
		strcat(aData, ADR('Engine_Version;'));	WRITE_STRING(ADR(IN_CB.szEng_Motorversion),aData);	strcat(aData, ADR('$n'));	(* Engine Version *)
		strcat(aData, ADR('Trigger_Event;'));	WRITE_DINT(iPBC_Trigger,aData);						strcat(aData, ADR('$n'));	(* Trigger *)
		strcat(aData, ADR(strLine));																							(* ------------ *)

		DerString		:=	'';
		iSize_String	:=	SIZEOF(DerString);
		iPointer		:=	ADR(DerString);
		iPointer		:=	save_strcat(ADR(DerString), iSize_String, iPointer, aData);											(* write std. header *)
		iPointer		:=	save_strcat(ADR(DerString), iSize_String, iPointer, aH);											(* write spec. header *)
		iZeile			:=	0;																									(* reset lines *)
		iStep			:=	_DATA;																								(* next step *)

		tiMax	:= -T#24h;
		tiMin	:=	T#24h;
		bFilled	:=	TRUE;
		FOR iCnt:=0 TO iBufferSize-1 DO
			IF Buffer.timer[iCnt] = T#0ms THEN
				bFilled	:=	FALSE;
			ELSE
				tiMax := MAX(tiMax, Buffer.timer[iCnt]);
				tiMin := MIN(tiMin, Buffer.timer[iCnt]);
			END_IF
		END_FOR

		IF tiMax > T#23h59m59s AND tiMin < T#1s THEN								(* wenn Tagwechsel *)
			FOR iCnt:=0 TO iBufferSize-1 DO
				IF Buffer.timer[iCnt] <> T#0ms AND Buffer.timer[iCnt] < T#1h THEN	(* erhoehe alle niederen um 24Stunden *)
					Buffer.timer[iCnt]	:=	Buffer.timer[iCnt] + T#24h;
				END_IF
			END_FOR
		END_IF

		IF NOT bFilled THEN															(* find Index 1, if buffer is not filled *)
			FOR iCnt:=0 TO iBufferSize DO
				IF Buffer.timer[(iCnt_Cycle + iCnt) MOD (iBufferSize)] > T#0s THEN EXIT; END_IF
			END_FOR
			iIdx1	:=	(iCnt_Cycle  + iCnt) MOD (iBufferSize);
		ELSE
			iIdx1	:=	(iCnt_Cycle ) MOD (iBufferSize);
		END_IF

(** 4.5: fill data string with data *)
	_DATA:
		FOR iAccel := 0 TO 2 DO																							(* write accelerator *)
		szData	:=	'';																										(* delete previous data line *)
		iIdx	:=	(iCnt_Cycle + iZeile) MOD (iBufferSize);																(* calculate ring buffer index *)
		iIdx10	:=	((iCnt_Cycle - (iCnt_Cycle MOD 10) +10 )/10 + UDINT_TO_INT((iZeile)/10)) MOD (iBufferSize/10);			(* calculate small ring buffer index *)
		bSCD_Ena:=	Buffer.timer[iIdx] > T#0s;
		IF bSCD_Ena THEN	WRITE_REAL(DINT_TO_REAL(TIME_TO_DINT(Buffer.timer[iIdx] - Buffer.timer[iIdx1]))/1000, 3, aData);				(* Time; *)
		ELSE				WRITE_REAL(0.0, 3, aData);																						(* 0.000; if empty *)
		END_IF
		FOR iCnt_B:=0 TO iBits_Max DO																										(* data bits *)
			IF Buffer.Bits[iCnt_B].used > 0 THEN WRITE_BIT(Buffer.Bits[iCnt_B].ucData[iIdx].0,aData);	END_IF									(* 0/1; *)
			IF Buffer.Bits[iCnt_B].used > 1 THEN WRITE_BIT(Buffer.Bits[iCnt_B].ucData[iIdx].1,aData);	END_IF									(* 0/1; *)
			IF Buffer.Bits[iCnt_B].used > 2 THEN WRITE_BIT(Buffer.Bits[iCnt_B].ucData[iIdx].2,aData);	END_IF									(* 0/1; *)
			IF Buffer.Bits[iCnt_B].used > 3 THEN WRITE_BIT(Buffer.Bits[iCnt_B].ucData[iIdx].3,aData);	END_IF									(* 0/1; *)
			IF Buffer.Bits[iCnt_B].used > 4 THEN WRITE_BIT(Buffer.Bits[iCnt_B].ucData[iIdx].4,aData);	END_IF									(* 0/1; *)
			IF Buffer.Bits[iCnt_B].used > 5 THEN WRITE_BIT(Buffer.Bits[iCnt_B].ucData[iIdx].5,aData);	END_IF									(* 0/1; *)
			IF Buffer.Bits[iCnt_B].used > 6 THEN WRITE_BIT(Buffer.Bits[iCnt_B].ucData[iIdx].6,aData);	END_IF									(* 0/1; *)
			IF Buffer.Bits[iCnt_B].used > 7 THEN WRITE_BIT(Buffer.Bits[iCnt_B].ucData[iIdx].7,aData);	END_IF									(* 0/1; *)
		END_FOR
		IF Buffer.iCnt_pattern > 0 THEN
			FOR iCnt:=0 TO Buffer.iCnt_pattern DO																								(* bit patterns *)
				FOR iCyl:=1 TO xEngType.NumberOfCylinder DO
					WRITE_BIT(UDINT_TO_BOOL(Buffer.pattern[iCnt].BitPattern[iIdx] AND REAL_TO_UDINT(2.0 ** (USINT_TO_REAL(iCyl)-1.0))),aData);		(* 0/1; *)
				END_FOR
			END_FOR
		END_IF
		FOR iCnt:=0 TO Buffer.iCnt_ui16_H DO																								(* task cycle data *)
			IF Buffer.ui16_H[iCnt].Signed THEN
				WRITE_REAL(INT_TO_REAL(UINT_TO_INT(Buffer.ui16_H[iCnt].Lo[iIdx]))/MAX(Buffer.ui16_H[iCnt].Co, 0.001), DECI(Buffer.ui16_H[iCnt].Co), aData);	(* Signed Value; *)
				WRITE_REAL(INT_TO_REAL(UINT_TO_INT(Buffer.ui16_H[iCnt].Hi[iIdx]))/MAX(Buffer.ui16_H[iCnt].Co, 0.001), DECI(Buffer.ui16_H[iCnt].Co), aData);	(* Signed Value; *)
			ELSE	WRITE_REAL(UINT_TO_REAL(Buffer.ui16_H[iCnt].Lo[iIdx])/MAX(Buffer.ui16_H[iCnt].Co, 0.001), DECI(Buffer.ui16_H[iCnt].Co), aData);			(* Unsigned Value; *)
					WRITE_REAL(UINT_TO_REAL(Buffer.ui16_H[iCnt].Hi[iIdx])/MAX(Buffer.ui16_H[iCnt].Co, 0.001), DECI(Buffer.ui16_H[iCnt].Co), aData);			(* Unsigned Value; *)
			END_IF
		END_FOR
		FOR iCnt:=0 TO Buffer.iCnt_ui16 DO																									(* engine cycle data *)
			IF Buffer.ui16[iCnt].Signed THEN
					WRITE_REAL(INT_TO_REAL(UINT_TO_INT(Buffer.ui16[iCnt].Data[iIdx]))/MAX(Buffer.ui16[iCnt].Co, 0.001), DECI(Buffer.ui16[iCnt].Co), aData);	(* Signed Value; *)
			ELSE	WRITE_REAL(UINT_TO_REAL(Buffer.ui16[iCnt].Data[iIdx])/MAX(Buffer.ui16[iCnt].Co, 0.001), DECI(Buffer.ui16[iCnt].Co), aData);				(* Unsigned Value; *)
			END_IF
		END_FOR
		FOR iCnt:=0 TO Buffer.iCnt_ui16_low DO																								(* slow changing data *)
			IF NOT bSCD_Ena THEN		WRITE_REAL(0.0, DECI(Buffer.ui16_low[iCnt].Co), aData);													(*0.0; if empty *)
			ELSIF Buffer.ui16_low[iCnt].Signed THEN
				WRITE_REAL(INT_TO_REAL(UINT_TO_INT(Buffer.ui16_low[iCnt].Data[iIdx10]))/MAX(Buffer.ui16_low[iCnt].Co, 0.001), DECI(Buffer.ui16_low[iCnt].Co), aData);	(* Signed Value; *)
			ELSE	WRITE_REAL(UINT_TO_REAL(Buffer.ui16_low[iCnt].Data[iIdx10])/MAX(Buffer.ui16_low[iCnt].Co, 0.001), DECI(Buffer.ui16_low[iCnt].Co), aData);			(* Unsigned Value; *)
			END_IF
		END_FOR
		strcat(aData, ADR('$n'));																											(* Return		*)
		iPointer	:=	save_strcat(ADR(DerString), iSize_String, iPointer, aData);															(* write data line *)
		iZeile	:=	MIN(iZeile+1,iBufferSize);																								(* increase line counter *)
		IF iZeile >= iBufferSize THEN
			iStep	:=	_FOOT;																												(* next step *)
			iAccel	:=	1000;																												(* break out of accelerator loop *)
		END_IF
		END_FOR
(** 4.6: fill data string with footer *)
	_FOOT:
		szData		:=	'';
		IF iPBC_Trigger = 1 THEN																						(* write SDT if engine trips *)
			szData		:=	'Slow down time; ';		WRITE_REAL(IN_CB.rSDT, 2, aData);	strcat(aData, ADR('s;$n'));			(* Slow down time;XXX;s; *)
		END_IF

		(**** ATD BEGIN ****)
		IF xEngType.Type9 THEN								//ATD experimental
			strcat(aData, ADR('<ATD>$n'));

			strcat(aData, ADR('logicMatrix_1; '));
			FOR iCnt:=0 TO iLogicSize_1 DO		WRITE_REAL(logicMatrix_1[iCnt], 0, aData);	END_FOR
			strcat(aData, ADR('$n'));

			strcat(aData, ADR('logicMatrix_2; '));
			FOR iCnt:=0 TO iLogicSize_2 DO		WRITE_REAL(logicMatrix_2[iCnt], 0, aData);	END_FOR
			strcat(aData, ADR('$n'));

			strcat(aData, ADR('splitVec; '));
			FOR iCnt:=0 TO iError_Channels DO	WRITE_REAL(LREAL_TO_REAL(splitVec[iCnt]), 0, aData);	END_FOR
			strcat(aData, ADR('$n'));

			FOR iCnt:=0 TO iError_Channels DO
				strcat(aData, ADR('FAM_struct.tCHL_'));
				WRITE_REAL(INT_TO_REAL(iCnt), 0, aData);
				FOR iCnt2:=0 TO iError_Depth DO	WRITE_REAL(USINT_TO_REAL(FAM_struct.tCHL[iCnt].chl[iCnt2]), 0, aData);	END_FOR
				strcat(aData, ADR('$n'));
			END_FOR

			strcat(aData, ADR('FAM_struct.mcc; '));
			FOR iCnt:=0 TO iError_Channels DO	WRITE_REAL(FAM_struct.mcc[iCnt], 4, aData);	END_FOR
			strcat(aData, ADR('$n'));

			strcat(aData, ADR('FAM_struct.cost_repair; '));
			FOR iCnt:=0 TO iError_Channels DO	WRITE_REAL(LREAL_TO_REAL(FAM_struct.cost_repair[iCnt]), 0, aData);	END_FOR
			strcat(aData, ADR('$n'));

			strcat(aData, ADR('FAM_struct.cost_not_repair; '));
			FOR iCnt:=0 TO iError_Channels DO	WRITE_REAL(LREAL_TO_REAL(FAM_struct.cost_not_repair[iCnt]), 0, aData);	END_FOR
			strcat(aData, ADR('$n'));

			strcat(aData, ADR('Pr_Knck_TH_MDN; '));				WRITE_REAL(FDT_value.Pr_Knck_TH_MDN,			2, aData);	strcat(aData, ADR('$n'));
			strcat(aData, ADR('Pr_Knck_TH_MDN_CNT; '));			WRITE_REAL(FDT_value.Pr_Knck_TH_MDN_CNT,		0, aData);	strcat(aData, ADR('$n'));

			strcat(aData, ADR('Pr_49bTDC_TH_MDN; '));			WRITE_REAL(FDT_value.Pr_49bTDC_TH_MDN,			2, aData);	strcat(aData, ADR('$n'));
			strcat(aData, ADR('Pr_49bTDC_TH_MDN_CNT; '));		WRITE_REAL(FDT_value.Pr_49bTDC_TH_MDN_CNT,		0, aData);	strcat(aData, ADR('$n'));

			strcat(aData, ADR('Pr_49aTDC_TH_MDN; '));			WRITE_REAL(FDT_value.Pr_49aTDC_TH_MDN,			2, aData);	strcat(aData, ADR('$n'));
			strcat(aData, ADR('Pr_49aTDC_TH_MDN_CNT; '));		WRITE_REAL(FDT_value.Pr_49aTDC_TH_MDN_CNT,		0, aData);	strcat(aData, ADR('$n'));

			strcat(aData, ADR('Pmax_TH_MDN; '));				WRITE_REAL(FDT_value.Pmax_TH_MDN,				2, aData);	strcat(aData, ADR('$n'));
			strcat(aData, ADR('Pmax_TH_MDN_CNT; '));			WRITE_REAL(FDT_value.Pmax_TH_MDN_CNT,			0, aData);	strcat(aData, ADR('$n'));

			strcat(aData, ADR('IMEP_TH_MDN; '));				WRITE_REAL(FDT_value.IMEP_TH_MDN,				2, aData);	strcat(aData, ADR('$n'));
			strcat(aData, ADR('IMEP_TH_MDN_CNT; '));			WRITE_REAL(FDT_value.IMEP_TH_MDN_CNT,			0, aData);	strcat(aData, ADR('$n'));

			strcat(aData, ADR('T_Exh_TH_MDN; '));				WRITE_REAL(FDT_value.T_Exh_TH_MDN,				2, aData);	strcat(aData, ADR('$n'));
			strcat(aData, ADR('T_Exh_TH_MDN_CNT; '));			WRITE_REAL(FDT_value.T_Exh_TH_MDN_CNT,			0, aData);	strcat(aData, ADR('$n'));

			strcat(aData, ADR('IT_TH_MDN; '));					WRITE_REAL(FDT_value.IT_TH_MDN,					2, aData);	strcat(aData, ADR('$n'));
			strcat(aData, ADR('IT_TH_MDN_CNT; '));				WRITE_REAL(FDT_value.IT_TH_MDN_CNT,				0, aData);	strcat(aData, ADR('$n'));

			strcat(aData, ADR('AI50_TH_MDN; '));				WRITE_REAL(FDT_value.AI50_TH_MDN,				2, aData);	strcat(aData, ADR('$n'));
			strcat(aData, ADR('AI50_TH_MDN_CNT; '));			WRITE_REAL(FDT_value.AI50_TH_MDN_CNT,			0, aData);	strcat(aData, ADR('$n'));

			strcat(aData, ADR('CA_PI_Duration_TH_MDN; '));		WRITE_REAL(FDT_value.CA_PI_Duration_TH_MDN,		2, aData);	strcat(aData, ADR('$n'));
			strcat(aData, ADR('CA_PI_Duration_TH_MDN_CNT; '));	WRITE_REAL(FDT_value.CA_PI_Duration_TH_MDN_CNT,	0, aData);	strcat(aData, ADR('$n'));

			strcat(aData, ADR('T_Rod_TH_MDN; '));				WRITE_REAL(FDT_value.T_Rod_TH_MDN,				2, aData);	strcat(aData, ADR('$n'));
			strcat(aData, ADR('T_Rod_TH_MDN_CNT; '));			WRITE_REAL(FDT_value.T_Rod_TH_MDN_CNT,			0, aData);	strcat(aData, ADR('$n'));

			strcat(aData, ADR('PBCSlowDriftCheck_CNT; '));		WRITE_REAL(FDT_value.PBCSlowDriftCheck_CNT,		0, aData);	strcat(aData, ADR('$n'));

			strcat(aData, ADR('integrator_increment; '));		WRITE_REAL(FDT_value.integrator_increment,		2, aData);	strcat(aData, ADR('$n'));
			strcat(aData, ADR('integrator_decay; '));			WRITE_REAL(FDT_value.integrator_decay,			2, aData);	strcat(aData, ADR('$n'));

			strcat(aData, ADR('filter_INT1_TH; '));				WRITE_REAL(FDT_value.filter_INT1_TH,			2, aData);	strcat(aData, ADR('$n'));

			(* P_Set *)
			strcat(aData, ADR('P_Set_Min_TH_s1_MAX; '));		WRITE_REAL(FDT_value.P_Set_Min_TH_s1_MAX,		0, aData);	strcat(aData, ADR('$n'));
			strcat(aData, ADR('P_Set_Min_TH_s1_CNT; '));		WRITE_REAL(FDT_value.P_Set_Min_TH_s1_CNT,		0, aData);	strcat(aData, ADR('$n'));
			strcat(aData, ADR('P_Set_Max_TH_s1_MAX; '));		WRITE_REAL(FDT_value.P_Set_Max_TH_s1_MAX,		0, aData);	strcat(aData, ADR('$n'));
			strcat(aData, ADR('P_Set_Max_TH_s1_CNT; '));		WRITE_REAL(FDT_value.P_Set_Max_TH_s1_CNT,		0, aData);	strcat(aData, ADR('$n'));
			(* P_Act *)
			strcat(aData, ADR('P_Act_Min_TH_REF; '));			WRITE_REAL(FDT_value.P_Act_Min_TH_REF,			2, aData);	strcat(aData, ADR('$n'));
			strcat(aData, ADR('P_Act_Min_TH_s1_MAX; '));		WRITE_REAL(FDT_value.P_Act_Min_TH_s1_MAX,		0, aData);	strcat(aData, ADR('$n'));
			strcat(aData, ADR('P_Act_Min_TH_REF_CNT; '));		WRITE_REAL(FDT_value.P_Act_Min_TH_REF_CNT,		0, aData);	strcat(aData, ADR('$n'));
			strcat(aData, ADR('P_Act_Min_TH_s1_CNT; '));		WRITE_REAL(FDT_value.P_Act_Min_TH_s1_CNT,		0, aData);	strcat(aData, ADR('$n'));
			strcat(aData, ADR('P_Act_Max_TH_REF; '));			WRITE_REAL(FDT_value.P_Act_Max_TH_REF,			2, aData);	strcat(aData, ADR('$n'));
			strcat(aData, ADR('P_Act_Max_TH_s1_MAX; '));		WRITE_REAL(FDT_value.P_Act_Max_TH_s1_MAX,		0, aData);	strcat(aData, ADR('$n'));
			strcat(aData, ADR('P_Act_Max_TH_REF_CNT; '));		WRITE_REAL(FDT_value.P_Act_Max_TH_REF_CNT,		0, aData);	strcat(aData, ADR('$n'));
			strcat(aData, ADR('P_Act_Max_TH_s1_CNT; '));		WRITE_REAL(FDT_value.P_Act_Max_TH_s1_CNT,		0, aData);	strcat(aData, ADR('$n'));

			(* P2s_A *)
			strcat(aData, ADR('Pr_P2s_A_Min_TH_REF; '));		WRITE_REAL(FDT_value.Pr_P2s_A_Min_TH_REF,		1, aData);	strcat(aData, ADR('$n'));
			strcat(aData, ADR('Pr_P2s_A_Min_TH_s1_MAX; '));		WRITE_REAL(FDT_value.Pr_P2s_A_Min_TH_s1_MAX,	0, aData);	strcat(aData, ADR('$n'));
			strcat(aData, ADR('Pr_P2s_A_Min_TH_REF_CNT; '));	WRITE_REAL(FDT_value.Pr_P2s_A_Min_TH_REF_CNT,	0, aData);	strcat(aData, ADR('$n'));
			strcat(aData, ADR('Pr_P2s_A_Min_TH_s1_CNT; '));		WRITE_REAL(FDT_value.Pr_P2s_A_Min_TH_s1_CNT,	0, aData);	strcat(aData, ADR('$n'));
			strcat(aData, ADR('Pr_P2s_A_Max_TH_REF; '));		WRITE_REAL(FDT_value.Pr_P2s_A_Max_TH_REF,		1, aData);	strcat(aData, ADR('$n'));
			strcat(aData, ADR('Pr_P2s_A_Max_TH_s1_MAX; '));		WRITE_REAL(FDT_value.Pr_P2s_A_Max_TH_s1_MAX,	0, aData);	strcat(aData, ADR('$n'));
			strcat(aData, ADR('Pr_P2s_A_Max_TH_REF_CNT; '));	WRITE_REAL(FDT_value.Pr_P2s_A_Max_TH_REF_CNT,	0, aData);	strcat(aData, ADR('$n'));
			strcat(aData, ADR('Pr_P2s_A_Max_TH_s1_CNT; '));		WRITE_REAL(FDT_value.Pr_P2s_A_Max_TH_s1_CNT,	0, aData);	strcat(aData, ADR('$n'));

			(* P2s_B *)
			strcat(aData, ADR('Pr_P2s_B_Min_TH_REF; '));		WRITE_REAL(FDT_value.Pr_P2s_B_Min_TH_REF,		1, aData);	strcat(aData, ADR('$n'));
			strcat(aData, ADR('Pr_P2s_B_Min_TH_s1_MAX; '));		WRITE_REAL(FDT_value.Pr_P2s_B_Min_TH_s1_MAX,	0, aData);	strcat(aData, ADR('$n'));
			strcat(aData, ADR('Pr_P2s_B_Min_TH_REF_CNT; '));	WRITE_REAL(FDT_value.Pr_P2s_B_Min_TH_REF_CNT,	0, aData);	strcat(aData, ADR('$n'));
			strcat(aData, ADR('Pr_P2s_B_Min_TH_s1_CNT; '));		WRITE_REAL(FDT_value.Pr_P2s_B_Min_TH_s1_CNT,	0, aData);	strcat(aData, ADR('$n'));
			strcat(aData, ADR('Pr_P2s_B_Max_TH_REF; '));		WRITE_REAL(FDT_value.Pr_P2s_B_Max_TH_REF,		1, aData);	strcat(aData, ADR('$n'));
			strcat(aData, ADR('Pr_P2s_B_Max_TH_s1_MAX; '));		WRITE_REAL(FDT_value.Pr_P2s_B_Max_TH_s1_MAX,	0, aData);	strcat(aData, ADR('$n'));
			strcat(aData, ADR('Pr_P2s_B_Max_TH_REF_CNT; '));	WRITE_REAL(FDT_value.Pr_P2s_B_Max_TH_REF_CNT,	0, aData);	strcat(aData, ADR('$n'));
			strcat(aData, ADR('Pr_P2s_B_Max_TH_s1_CNT; '));		WRITE_REAL(FDT_value.Pr_P2s_B_Max_TH_s1_CNT,	0, aData);	strcat(aData, ADR('$n'));

			(* Pr_Leanox *)
			strcat(aData, ADR('Pr_Leanox_Set_Min_TH_s1_MAX; '));	WRITE_REAL(FDT_value.Pr_Leanox_Set_Min_TH_s1_MAX,	0, aData);	strcat(aData, ADR('$n'));
			strcat(aData, ADR('Pr_Leanox_Set_Min_TH_s1_CNT; '));	WRITE_REAL(FDT_value.Pr_Leanox_Set_Min_TH_s1_CNT,	0, aData);	strcat(aData, ADR('$n'));
			strcat(aData, ADR('Pr_Leanox_Set_Max_TH_s1_MAX; '));	WRITE_REAL(FDT_value.Pr_Leanox_Set_Max_TH_s1_MAX,	0, aData);	strcat(aData, ADR('$n'));
			strcat(aData, ADR('Pr_Leanox_Set_Max_TH_s1_CNT; '));	WRITE_REAL(FDT_value.Pr_Leanox_Set_Max_TH_s1_CNT,	0, aData);	strcat(aData, ADR('$n'));

			(* GR_Set *)
			strcat(aData, ADR('Pr_GR_Set_Min_TH_s1_MAX; '));		WRITE_REAL(FDT_value.Pr_GR_Set_Min_TH_s1_MAX,	0, aData);	strcat(aData, ADR('$n'));
			strcat(aData, ADR('Pr_GR_Set_Min_TH_s1_CNT; '));		WRITE_REAL(FDT_value.Pr_GR_Set_Min_TH_s1_CNT,	0, aData);	strcat(aData, ADR('$n'));
			strcat(aData, ADR('Pr_GR_Set_Max_TH_s1_MAX; '));		WRITE_REAL(FDT_value.Pr_GR_Set_Max_TH_s1_MAX,	0, aData);	strcat(aData, ADR('$n'));
			strcat(aData, ADR('Pr_GR_Set_Max_TH_s1_CNT; '));		WRITE_REAL(FDT_value.Pr_GR_Set_Max_TH_s1_CNT,	0, aData);	strcat(aData, ADR('$n'));
			(* GR_Act *)
			strcat(aData, ADR('Pr_GR_Act_Min_TH_REF; '));			WRITE_REAL(FDT_value.Pr_GR_Act_Min_TH_REF,		1, aData);	strcat(aData, ADR('$n'));
			strcat(aData, ADR('Pr_GR_Act_Min_TH_s1_MAX; '));		WRITE_REAL(FDT_value.Pr_GR_Act_Min_TH_s1_MAX,	0, aData);	strcat(aData, ADR('$n'));
			strcat(aData, ADR('Pr_GR_Act_Min_TH_REF_CNT; '));		WRITE_REAL(FDT_value.Pr_GR_Act_Min_TH_REF_CNT,	0, aData);	strcat(aData, ADR('$n'));
			strcat(aData, ADR('Pr_GR_Act_Min_TH_s1_CNT; '));		WRITE_REAL(FDT_value.Pr_GR_Act_Min_TH_s1_CNT,	0, aData);	strcat(aData, ADR('$n'));
			strcat(aData, ADR('Pr_GR_Act_Max_TH_REF; '));			WRITE_REAL(FDT_value.Pr_GR_Act_Max_TH_REF,		1, aData);	strcat(aData, ADR('$n'));
			strcat(aData, ADR('Pr_GR_Act_Max_TH_s1_MAX; '));		WRITE_REAL(FDT_value.Pr_GR_Act_Max_TH_s1_MAX,	0, aData);	strcat(aData, ADR('$n'));
			strcat(aData, ADR('Pr_GR_Act_Max_TH_REF_CNT; '));		WRITE_REAL(FDT_value.Pr_GR_Act_Max_TH_REF_CNT,	0, aData);	strcat(aData, ADR('$n'));
			strcat(aData, ADR('Pr_GR_Act_Max_TH_s1_CNT; '));		WRITE_REAL(FDT_value.Pr_GR_Act_Max_TH_s1_CNT,	0, aData);	strcat(aData, ADR('$n'));

			(* PC_Set *)
			strcat(aData, ADR('Pr_PC_Set_Min_TH_s1_MAX; '));		WRITE_REAL(FDT_value.Pr_PC_Set_Min_TH_s1_MAX,	0, aData);	strcat(aData, ADR('$n'));
			strcat(aData, ADR('Pr_PC_Set_Min_TH_s1_CNT; '));		WRITE_REAL(FDT_value.Pr_PC_Set_Min_TH_s1_CNT,	0, aData);	strcat(aData, ADR('$n'));
			strcat(aData, ADR('Pr_PC_Set_Max_TH_s1_MAX; '));		WRITE_REAL(FDT_value.Pr_PC_Set_Max_TH_s1_MAX,	0, aData);	strcat(aData, ADR('$n'));
			strcat(aData, ADR('Pr_PC_Set_Max_TH_s1_CNT; '));		WRITE_REAL(FDT_value.Pr_PC_Set_Max_TH_s1_CNT,	0, aData);	strcat(aData, ADR('$n'));
			(* PC_Act *)
			strcat(aData, ADR('Pr_PC_Act_Min_TH_REF; '));			WRITE_REAL(FDT_value.Pr_PC_Act_Min_TH_REF,		1, aData);	strcat(aData, ADR('$n'));
			strcat(aData, ADR('Pr_PC_Act_Min_TH_s1_MAX; '));		WRITE_REAL(FDT_value.Pr_PC_Act_Min_TH_s1_MAX,	0, aData);	strcat(aData, ADR('$n'));
			strcat(aData, ADR('Pr_PC_Act_Min_TH_REF_CNT; '));		WRITE_REAL(FDT_value.Pr_PC_Act_Min_TH_REF_CNT,	0, aData);	strcat(aData, ADR('$n'));
			strcat(aData, ADR('Pr_PC_Act_Min_TH_s1_CNT; '));		WRITE_REAL(FDT_value.Pr_PC_Act_Min_TH_s1_CNT,	0, aData);	strcat(aData, ADR('$n'));
			strcat(aData, ADR('Pr_PC_Act_Max_TH_REF; '));			WRITE_REAL(FDT_value.Pr_PC_Act_Max_TH_REF,		1, aData);	strcat(aData, ADR('$n'));
			strcat(aData, ADR('Pr_PC_Act_Max_TH_s1_MAX; '));		WRITE_REAL(FDT_value.Pr_PC_Act_Max_TH_s1_MAX,	0, aData);	strcat(aData, ADR('$n'));
			strcat(aData, ADR('Pr_PC_Act_Max_TH_REF_CNT; '));		WRITE_REAL(FDT_value.Pr_PC_Act_Max_TH_REF_CNT,	0, aData);	strcat(aData, ADR('$n'));
			strcat(aData, ADR('Pr_PC_Act_Max_TH_s1_CNT; '));		WRITE_REAL(FDT_value.Pr_PC_Act_Max_TH_s1_CNT,	0, aData);	strcat(aData, ADR('$n'));

			(* Pos_CBV *)
			strcat(aData, ADR('Pos_CBV_Set_Min_TH_s1_MAX; '));	WRITE_REAL(FDT_value.Pos_CBV_Set_Min_TH_s1_MAX,	1, aData);	strcat(aData, ADR('$n'));
			strcat(aData, ADR('Pos_CBV_Set_Max_TH_s1_MAX; '));	WRITE_REAL(FDT_value.Pos_CBV_Set_Max_TH_s1_MAX,	1, aData);	strcat(aData, ADR('$n'));
			strcat(aData, ADR('Pos_CBV_Set_Min_TH_s1_CNT; '));	WRITE_REAL(FDT_value.Pos_CBV_Set_Min_TH_s1_CNT,	0, aData);	strcat(aData, ADR('$n'));
			strcat(aData, ADR('Pos_CBV_Set_Max_TH_s1_CNT; '));	WRITE_REAL(FDT_value.Pos_CBV_Set_Max_TH_s1_CNT,	0, aData);	strcat(aData, ADR('$n'));

			strcat(aData, ADR('Pos_CBV_A1_Min_TH_REF; '));		WRITE_REAL(FDT_value.Pos_CBV_A1_Min_TH_REF,		2, aData);	strcat(aData, ADR('$n'));
			strcat(aData, ADR('Pos_CBV_A1_Min_TH_s1_MAX; '));	WRITE_REAL(FDT_value.Pos_CBV_A1_Min_TH_s1_MAX,	1, aData);	strcat(aData, ADR('$n'));
			strcat(aData, ADR('Pos_CBV_A1_Min_TH_REF_CNT; '));	WRITE_REAL(FDT_value.Pos_CBV_A1_Min_TH_REF_CNT,	0, aData);	strcat(aData, ADR('$n'));
			strcat(aData, ADR('Pos_CBV_A1_Min_TH_s1_CNT; '));	WRITE_REAL(FDT_value.Pos_CBV_A1_Min_TH_s1_CNT,	0, aData);	strcat(aData, ADR('$n'));
			strcat(aData, ADR('Pos_CBV_A1_Max_TH_REF; '));		WRITE_REAL(FDT_value.Pos_CBV_A1_Max_TH_REF,		2, aData);	strcat(aData, ADR('$n'));
			strcat(aData, ADR('Pos_CBV_A1_Max_TH_s1_MAX; '));	WRITE_REAL(FDT_value.Pos_CBV_A1_Max_TH_s1_MAX,	1, aData);	strcat(aData, ADR('$n'));
			strcat(aData, ADR('Pos_CBV_A1_Max_TH_REF_CNT; '));	WRITE_REAL(FDT_value.Pos_CBV_A1_Max_TH_REF_CNT,	0, aData);	strcat(aData, ADR('$n'));
			strcat(aData, ADR('Pos_CBV_A1_Max_TH_s1_CNT; '));	WRITE_REAL(FDT_value.Pos_CBV_A1_Max_TH_s1_CNT,	0, aData);	strcat(aData, ADR('$n'));

			strcat(aData, ADR('Pos_CBV_B1_Min_TH_REF; '));		WRITE_REAL(FDT_value.Pos_CBV_B1_Min_TH_REF,		2, aData);	strcat(aData, ADR('$n'));
			strcat(aData, ADR('Pos_CBV_B1_Min_TH_s1_MAX; '));	WRITE_REAL(FDT_value.Pos_CBV_B1_Min_TH_s1_MAX,	1, aData);	strcat(aData, ADR('$n'));
			strcat(aData, ADR('Pos_CBV_B1_Min_TH_REF_CNT; '));	WRITE_REAL(FDT_value.Pos_CBV_B1_Min_TH_REF_CNT,	0, aData);	strcat(aData, ADR('$n'));
			strcat(aData, ADR('Pos_CBV_B1_Min_TH_s1_CNT; '));	WRITE_REAL(FDT_value.Pos_CBV_B1_Min_TH_s1_CNT,	0, aData);	strcat(aData, ADR('$n'));
			strcat(aData, ADR('Pos_CBV_B1_Max_TH_REF; '));		WRITE_REAL(FDT_value.Pos_CBV_B1_Max_TH_REF,		2, aData);	strcat(aData, ADR('$n'));
			strcat(aData, ADR('Pos_CBV_B1_Max_TH_s1_MAX; '));	WRITE_REAL(FDT_value.Pos_CBV_B1_Max_TH_s1_MAX,	1, aData);	strcat(aData, ADR('$n'));
			strcat(aData, ADR('Pos_CBV_B1_Max_TH_REF_CNT; '));	WRITE_REAL(FDT_value.Pos_CBV_B1_Max_TH_REF_CNT,	0, aData);	strcat(aData, ADR('$n'));
			strcat(aData, ADR('Pos_CBV_B1_Max_TH_s1_CNT; '));	WRITE_REAL(FDT_value.Pos_CBV_B1_Max_TH_s1_CNT,	0, aData);	strcat(aData, ADR('$n'));

			(* Speed *)
			strcat(aData, ADR('Speed_NOM; '));					WRITE_REAL(FDT_value.Speed_NOM,					0, aData);	strcat(aData, ADR('$n'));
			strcat(aData, ADR('Speed_Min_TH_NOM; '));			WRITE_REAL(FDT_value.Speed_Min_TH_NOM,			1, aData);	strcat(aData, ADR('$n'));
			strcat(aData, ADR('Speed_Min_TH_s1_MAX; '));		WRITE_REAL(FDT_value.Speed_Min_TH_s1_MAX,		0, aData);	strcat(aData, ADR('$n'));
			strcat(aData, ADR('Speed_Min_TH_NOM_CNT; '));		WRITE_REAL(FDT_value.Speed_Min_TH_NOM_CNT,		0, aData);	strcat(aData, ADR('$n'));
			strcat(aData, ADR('Speed_Min_TH_s1_CNT; '));		WRITE_REAL(FDT_value.Speed_Min_TH_s1_CNT,		0, aData);	strcat(aData, ADR('$n'));
			strcat(aData, ADR('Speed_Max_TH_NOM; '));			WRITE_REAL(FDT_value.Speed_Max_TH_NOM,			1, aData);	strcat(aData, ADR('$n'));
			strcat(aData, ADR('Speed_Max_TH_s1_MAX; '));		WRITE_REAL(FDT_value.Speed_Max_TH_s1_MAX,		0, aData);	strcat(aData, ADR('$n'));
			strcat(aData, ADR('Speed_Max_TH_NOM_CNT; '));		WRITE_REAL(FDT_value.Speed_Max_TH_NOM_CNT,		0, aData);	strcat(aData, ADR('$n'));
			strcat(aData, ADR('Speed_Max_TH_s1_CNT; '));		WRITE_REAL(FDT_value.Speed_Max_TH_s1_CNT,		0, aData);	strcat(aData, ADR('$n'));

			(* T2s *)
			strcat(aData, ADR('T_T2s_NOM; '));					WRITE_REAL(FDT_value.T_T2s_NOM,					0, aData);	strcat(aData, ADR('$n'));
			strcat(aData, ADR('T_T2s_TH_NOM; '));				WRITE_REAL(FDT_value.T_T2s_TH_NOM,				1, aData);	strcat(aData, ADR('$n'));
			strcat(aData, ADR('T_T2s_TH_s1_MAX; '));			WRITE_REAL(FDT_value.T_T2s_TH_s1_MAX,			0, aData);	strcat(aData, ADR('$n'));
			strcat(aData, ADR('T_T2s_TH_NOM_CNT; '));			WRITE_REAL(FDT_value.T_T2s_TH_NOM_CNT,			0, aData);	strcat(aData, ADR('$n'));
			strcat(aData, ADR('T_T2s_TH_s1_CNT; '));			WRITE_REAL(FDT_value.T_T2s_TH_s1_CNT,			0, aData);	strcat(aData, ADR('$n'));

			(* Lam_Set *)
			strcat(aData, ADR('Lam_Set_Min_NOM; '));			WRITE_REAL(FDT_value.Lam_Set_Min_NOM,			0, aData);	strcat(aData, ADR('$n'));
			strcat(aData, ADR('Lam_Set_Min_TH_NOM; '));			WRITE_REAL(FDT_value.Lam_Set_Min_TH_NOM,		2, aData);	strcat(aData, ADR('$n'));
			strcat(aData, ADR('Lam_Set_Min_TH_s1_MAX; '));		WRITE_REAL(FDT_value.Lam_Set_Min_TH_s1_MAX,		0, aData);	strcat(aData, ADR('$n'));
			strcat(aData, ADR('Lam_Set_Min_TH_NOM_CNT; '));		WRITE_REAL(FDT_value.Lam_Set_Min_TH_NOM_CNT,	0, aData);	strcat(aData, ADR('$n'));
			strcat(aData, ADR('Lam_Set_Min_TH_s1_CNT; '));		WRITE_REAL(FDT_value.Lam_Set_Min_TH_s1_CNT,		0, aData);	strcat(aData, ADR('$n'));
			strcat(aData, ADR('Lam_Set_Max_NOM; '));			WRITE_REAL(FDT_value.Lam_Set_Max_NOM,			0, aData);	strcat(aData, ADR('$n'));
			strcat(aData, ADR('Lam_Set_Max_TH_NOM; '));			WRITE_REAL(FDT_value.Lam_Set_Max_TH_NOM,		2, aData);	strcat(aData, ADR('$n'));
			strcat(aData, ADR('Lam_Set_Max_TH_s1_MAX; '));		WRITE_REAL(FDT_value.Lam_Set_Max_TH_s1_MAX,		0, aData);	strcat(aData, ADR('$n'));
			strcat(aData, ADR('Lam_Set_Max_TH_NOM_CNT; '));		WRITE_REAL(FDT_value.Lam_Set_Max_TH_NOM_CNT,	0, aData);	strcat(aData, ADR('$n'));
			strcat(aData, ADR('Lam_Set_Max_TH_s1_CNT; '));		WRITE_REAL(FDT_value.Lam_Set_Max_TH_s1_CNT,		0, aData);	strcat(aData, ADR('$n'));

			(* U_L1L2 *)
			strcat(aData, ADR('U_L1L2_Min_NOM; '));				WRITE_REAL(FDT_value.U_L1L2_Min_NOM,			0, aData);	strcat(aData, ADR('$n'));
			strcat(aData, ADR('U_L1L2_Min_TH_NOM; '));			WRITE_REAL(FDT_value.U_L1L2_Min_TH_NOM,			1, aData);	strcat(aData, ADR('$n'));
			strcat(aData, ADR('U_L1L2_Min_TH_s1_MAX; '));		WRITE_REAL(FDT_value.U_L1L2_Min_TH_s1_MAX,		0, aData);	strcat(aData, ADR('$n'));
			strcat(aData, ADR('U_L1L2_Min_TH_NOM_CNT; '));		WRITE_REAL(FDT_value.U_L1L2_Min_TH_NOM_CNT,		0, aData);	strcat(aData, ADR('$n'));
			strcat(aData, ADR('U_L1L2_Min_TH_s1_CNT; '));		WRITE_REAL(FDT_value.U_L1L2_Min_TH_s1_CNT,		0, aData);	strcat(aData, ADR('$n'));
			strcat(aData, ADR('U_L1L2_Max_NOM; '));				WRITE_REAL(FDT_value.U_L1L2_Max_NOM,			0, aData);	strcat(aData, ADR('$n'));
			strcat(aData, ADR('U_L1L2_Max_TH_NOM; '));			WRITE_REAL(FDT_value.U_L1L2_Max_TH_NOM,			1, aData);	strcat(aData, ADR('$n'));
			strcat(aData, ADR('U_L1L2_Max_TH_s1_MAX; '));		WRITE_REAL(FDT_value.U_L1L2_Max_TH_s1_MAX,		0, aData);	strcat(aData, ADR('$n'));
			strcat(aData, ADR('U_L1L2_Max_TH_NOM_CNT; '));		WRITE_REAL(FDT_value.U_L1L2_Max_TH_NOM_CNT,		0, aData);	strcat(aData, ADR('$n'));
			strcat(aData, ADR('U_L1L2_Max_TH_s1_CNT; '));		WRITE_REAL(FDT_value.U_L1L2_Max_TH_s1_CNT,		0, aData);	strcat(aData, ADR('$n'));

			(* U_L2L3 *)
			strcat(aData, ADR('U_L2L3_Min_NOM; '));				WRITE_REAL(FDT_value.U_L2L3_Min_NOM,			0, aData);	strcat(aData, ADR('$n'));
			strcat(aData, ADR('U_L2L3_Min_TH_NOM; '));			WRITE_REAL(FDT_value.U_L2L3_Min_TH_NOM,			1, aData);	strcat(aData, ADR('$n'));
			strcat(aData, ADR('U_L2L3_Min_TH_s1_MAX; '));		WRITE_REAL(FDT_value.U_L2L3_Min_TH_s1_MAX,		0, aData);	strcat(aData, ADR('$n'));
			strcat(aData, ADR('U_L2L3_Min_TH_NOM_CNT; '));		WRITE_REAL(FDT_value.U_L2L3_Min_TH_NOM_CNT,		0, aData);	strcat(aData, ADR('$n'));
			strcat(aData, ADR('U_L2L3_Min_TH_s1_CNT; '));		WRITE_REAL(FDT_value.U_L2L3_Min_TH_s1_CNT,		0, aData);	strcat(aData, ADR('$n'));
			strcat(aData, ADR('U_L2L3_Max_NOM; '));				WRITE_REAL(FDT_value.U_L2L3_Max_NOM,			0, aData);	strcat(aData, ADR('$n'));
			strcat(aData, ADR('U_L2L3_Max_TH_NOM; '));			WRITE_REAL(FDT_value.U_L2L3_Max_TH_NOM,			1, aData);	strcat(aData, ADR('$n'));
			strcat(aData, ADR('U_L2L3_Max_TH_s1_MAX; '));		WRITE_REAL(FDT_value.U_L2L3_Max_TH_s1_MAX,		0, aData);	strcat(aData, ADR('$n'));
			strcat(aData, ADR('U_L2L3_Max_TH_NOM_CNT; '));		WRITE_REAL(FDT_value.U_L2L3_Max_TH_NOM_CNT,		0, aData);	strcat(aData, ADR('$n'));
			strcat(aData, ADR('U_L2L3_Max_TH_s1_CNT; '));		WRITE_REAL(FDT_value.U_L2L3_Max_TH_s1_CNT,		0, aData);	strcat(aData, ADR('$n'));

			(* U_L3L1 *)
			strcat(aData, ADR('U_L3L1_Min_NOM; '));				WRITE_REAL(FDT_value.U_L3L1_Min_NOM,			0, aData);	strcat(aData, ADR('$n'));
			strcat(aData, ADR('U_L3L1_Min_TH_NOM; '));			WRITE_REAL(FDT_value.U_L3L1_Min_TH_NOM,			1, aData);	strcat(aData, ADR('$n'));
			strcat(aData, ADR('U_L3L1_Min_TH_s1_MAX; '));		WRITE_REAL(FDT_value.U_L3L1_Min_TH_s1_MAX,		0, aData);	strcat(aData, ADR('$n'));
			strcat(aData, ADR('U_L3L1_Min_TH_NOM_CNT; '));		WRITE_REAL(FDT_value.U_L3L1_Min_TH_NOM_CNT,		0, aData);	strcat(aData, ADR('$n'));
			strcat(aData, ADR('U_L3L1_Min_TH_s1_CNT; '));		WRITE_REAL(FDT_value.U_L3L1_Min_TH_s1_CNT,		0, aData);	strcat(aData, ADR('$n'));
			strcat(aData, ADR('U_L3L1_Max_NOM; '));				WRITE_REAL(FDT_value.U_L3L1_Max_NOM,			0, aData);	strcat(aData, ADR('$n'));
			strcat(aData, ADR('U_L3L1_Max_TH_NOM; '));			WRITE_REAL(FDT_value.U_L3L1_Max_TH_NOM,			1, aData);	strcat(aData, ADR('$n'));
			strcat(aData, ADR('U_L3L1_Max_TH_s1_MAX; '));		WRITE_REAL(FDT_value.U_L3L1_Max_TH_s1_MAX,		0, aData);	strcat(aData, ADR('$n'));
			strcat(aData, ADR('U_L3L1_Max_TH_NOM_CNT; '));		WRITE_REAL(FDT_value.U_L3L1_Max_TH_NOM_CNT,		0, aData);	strcat(aData, ADR('$n'));
			strcat(aData, ADR('U_L3L1_Max_TH_s1_CNT; '));		WRITE_REAL(FDT_value.U_L3L1_Max_TH_s1_CNT,		0, aData);	strcat(aData, ADR('$n'));

			(* I_L1 *)
			strcat(aData, ADR('I_L1_Min_NOM; '));				WRITE_REAL(FDT_value.I_L1_Min_NOM,				0, aData);	strcat(aData, ADR('$n'));
			strcat(aData, ADR('I_L1_Min_TH_NOM; '));			WRITE_REAL(FDT_value.I_L1_Min_TH_NOM,			3, aData);	strcat(aData, ADR('$n'));
			strcat(aData, ADR('I_L1_Min_TH_s1_MAX; '));			WRITE_REAL(FDT_value.I_L1_Min_TH_s1_MAX,		0, aData);	strcat(aData, ADR('$n'));
			strcat(aData, ADR('I_L1_Min_TH_NOM_CNT; '));		WRITE_REAL(FDT_value.I_L1_Min_TH_NOM_CNT,		0, aData);	strcat(aData, ADR('$n'));
			strcat(aData, ADR('I_L1_Min_TH_s1_CNT; '));			WRITE_REAL(FDT_value.I_L1_Min_TH_s1_CNT,		0, aData);	strcat(aData, ADR('$n'));
			strcat(aData, ADR('I_L1_Max_NOM; '));				WRITE_REAL(FDT_value.I_L1_Max_NOM,				0, aData);	strcat(aData, ADR('$n'));
			strcat(aData, ADR('I_L1_Max_TH_NOM; '));			WRITE_REAL(FDT_value.I_L1_Max_TH_NOM,			3, aData);	strcat(aData, ADR('$n'));
			strcat(aData, ADR('I_L1_Max_TH_s1_MAX; '));			WRITE_REAL(FDT_value.I_L1_Max_TH_s1_MAX,		0, aData);	strcat(aData, ADR('$n'));
			strcat(aData, ADR('I_L1_Max_TH_NOM_CNT; '));		WRITE_REAL(FDT_value.I_L1_Max_TH_NOM_CNT,		0, aData);	strcat(aData, ADR('$n'));
			strcat(aData, ADR('I_L1_Max_TH_s1_CNT; '));			WRITE_REAL(FDT_value.I_L1_Max_TH_s1_CNT,		0, aData);	strcat(aData, ADR('$n'));

			(* I_L2 *)
			strcat(aData, ADR('I_L2_Min_NOM; '));				WRITE_REAL(FDT_value.I_L2_Min_NOM,				0, aData);	strcat(aData, ADR('$n'));
			strcat(aData, ADR('I_L2_Min_TH_NOM; '));			WRITE_REAL(FDT_value.I_L2_Min_TH_NOM,			3, aData);	strcat(aData, ADR('$n'));
			strcat(aData, ADR('I_L2_Min_TH_s1_MAX; '));			WRITE_REAL(FDT_value.I_L2_Min_TH_s1_MAX,		0, aData);	strcat(aData, ADR('$n'));
			strcat(aData, ADR('I_L2_Min_TH_NOM_CNT; '));		WRITE_REAL(FDT_value.I_L2_Min_TH_NOM_CNT,		0, aData);	strcat(aData, ADR('$n'));
			strcat(aData, ADR('I_L2_Min_TH_s1_CNT; '));			WRITE_REAL(FDT_value.I_L2_Min_TH_s1_CNT,		0, aData);	strcat(aData, ADR('$n'));
			strcat(aData, ADR('I_L2_Max_NOM; '));				WRITE_REAL(FDT_value.I_L2_Max_NOM,				0, aData);	strcat(aData, ADR('$n'));
			strcat(aData, ADR('I_L2_Max_TH_NOM; '));			WRITE_REAL(FDT_value.I_L2_Max_TH_NOM,			3, aData);	strcat(aData, ADR('$n'));
			strcat(aData, ADR('I_L2_Max_TH_s1_MAX; '));			WRITE_REAL(FDT_value.I_L2_Max_TH_s1_MAX,		0, aData);	strcat(aData, ADR('$n'));
			strcat(aData, ADR('I_L2_Max_TH_NOM_CNT; '));		WRITE_REAL(FDT_value.I_L2_Max_TH_NOM_CNT,		0, aData);	strcat(aData, ADR('$n'));
			strcat(aData, ADR('I_L2_Max_TH_s1_CNT; '));			WRITE_REAL(FDT_value.I_L2_Max_TH_s1_CNT,		0, aData);	strcat(aData, ADR('$n'));

			(* I_L3 *)
			strcat(aData, ADR('I_L3_Min_NOM; '));				WRITE_REAL(FDT_value.I_L3_Min_NOM,				0, aData);	strcat(aData, ADR('$n'));
			strcat(aData, ADR('I_L3_Min_TH_NOM; '));			WRITE_REAL(FDT_value.I_L3_Min_TH_NOM,			3, aData);	strcat(aData, ADR('$n'));
			strcat(aData, ADR('I_L3_Min_TH_s1_MAX; '));			WRITE_REAL(FDT_value.I_L3_Min_TH_s1_MAX,		0, aData);	strcat(aData, ADR('$n'));
			strcat(aData, ADR('I_L3_Min_TH_NOM_CNT; '));		WRITE_REAL(FDT_value.I_L3_Min_TH_NOM_CNT,		0, aData);	strcat(aData, ADR('$n'));
			strcat(aData, ADR('I_L3_Min_TH_s1_CNT; '));			WRITE_REAL(FDT_value.I_L3_Min_TH_s1_CNT,		0, aData);	strcat(aData, ADR('$n'));
			strcat(aData, ADR('I_L3_Max_NOM; '));				WRITE_REAL(FDT_value.I_L3_Max_NOM,				0, aData);	strcat(aData, ADR('$n'));
			strcat(aData, ADR('I_L3_Max_TH_NOM; '));			WRITE_REAL(FDT_value.I_L3_Max_TH_NOM,			3, aData);	strcat(aData, ADR('$n'));
			strcat(aData, ADR('I_L3_Max_TH_s1_MAX; '));			WRITE_REAL(FDT_value.I_L3_Max_TH_s1_MAX,		0, aData);	strcat(aData, ADR('$n'));
			strcat(aData, ADR('I_L3_Max_TH_NOM_CNT; '));		WRITE_REAL(FDT_value.I_L3_Max_TH_NOM_CNT,		0, aData);	strcat(aData, ADR('$n'));
			strcat(aData, ADR('I_L3_Max_TH_s1_CNT; '));			WRITE_REAL(FDT_value.I_L3_Max_TH_s1_CNT,		0, aData);	strcat(aData, ADR('$n'));

			(* Q *)
			strcat(aData, ADR('Q_Min_NOM; '));					WRITE_REAL(FDT_value.Q_Min_NOM,					0, aData);	strcat(aData, ADR('$n'));
			strcat(aData, ADR('Q_Min_TH_NOM; '));				WRITE_REAL(FDT_value.Q_Min_TH_NOM,				1, aData);	strcat(aData, ADR('$n'));
			strcat(aData, ADR('Q_Min_TH_s1_MAX; '));			WRITE_REAL(FDT_value.Q_Min_TH_s1_MAX,			0, aData);	strcat(aData, ADR('$n'));
			strcat(aData, ADR('Q_Min_TH_NOM_CNT; '));			WRITE_REAL(FDT_value.Q_Min_TH_NOM_CNT,			0, aData);	strcat(aData, ADR('$n'));
			strcat(aData, ADR('Q_Min_TH_s1_CNT; '));			WRITE_REAL(FDT_value.Q_Min_TH_s1_CNT,			0, aData);	strcat(aData, ADR('$n'));
			strcat(aData, ADR('Q_Max_NOM; '));					WRITE_REAL(FDT_value.Q_Max_NOM,					0, aData);	strcat(aData, ADR('$n'));
			strcat(aData, ADR('Q_Max_TH_NOM; '));				WRITE_REAL(FDT_value.Q_Max_TH_NOM,				1, aData);	strcat(aData, ADR('$n'));
			strcat(aData, ADR('Q_Max_TH_s1_MAX; '));			WRITE_REAL(FDT_value.Q_Max_TH_s1_MAX,			0, aData);	strcat(aData, ADR('$n'));
			strcat(aData, ADR('Q_Max_TH_NOM_CNT; '));			WRITE_REAL(FDT_value.Q_Max_TH_NOM_CNT,			0, aData);	strcat(aData, ADR('$n'));
			strcat(aData, ADR('Q_Max_TH_s1_CNT; '));			WRITE_REAL(FDT_value.Q_Max_TH_s1_CNT,			0, aData);	strcat(aData, ADR('$n'));

			(* F *)
			strcat(aData, ADR('Freq_Min_NOM; '));				WRITE_REAL(FDT_value.Freq_Min_NOM,				0, aData);	strcat(aData, ADR('$n'));
			strcat(aData, ADR('Freq_Min_TH_NOM; '));			WRITE_REAL(FDT_value.Freq_Min_TH_NOM,			1, aData);	strcat(aData, ADR('$n'));
			strcat(aData, ADR('Freq_Min_TH_s1_MAX; '));			WRITE_REAL(FDT_value.Freq_Min_TH_s1_MAX,		0, aData);	strcat(aData, ADR('$n'));
			strcat(aData, ADR('Freq_Min_TH_NOM_CNT; '));		WRITE_REAL(FDT_value.Freq_Min_TH_NOM_CNT,		0, aData);	strcat(aData, ADR('$n'));
			strcat(aData, ADR('Freq_Min_TH_s1_CNT; '));			WRITE_REAL(FDT_value.Freq_Min_TH_s1_CNT,		0, aData);	strcat(aData, ADR('$n'));
			strcat(aData, ADR('Freq_Max_NOM; '));				WRITE_REAL(FDT_value.Freq_Max_NOM,				0, aData);	strcat(aData, ADR('$n'));
			strcat(aData, ADR('Freq_Max_TH_NOM; '));			WRITE_REAL(FDT_value.Freq_Max_TH_NOM,			1, aData);	strcat(aData, ADR('$n'));
			strcat(aData, ADR('Freq_Max_TH_s1_MAX; '));			WRITE_REAL(FDT_value.Freq_Max_TH_s1_MAX,		0, aData);	strcat(aData, ADR('$n'));
			strcat(aData, ADR('Freq_Max_TH_NOM_CNT; '));		WRITE_REAL(FDT_value.Freq_Max_TH_NOM_CNT,		0, aData);	strcat(aData, ADR('$n'));
			strcat(aData, ADR('Freq_Max_TH_s1_CNT; '));			WRITE_REAL(FDT_value.Freq_Max_TH_s1_CNT,		0, aData);	strcat(aData, ADR('$n'));

			(* CosPhi *)
			strcat(aData, ADR('CosPhi_Min_NOM; '));				WRITE_REAL(FDT_value.CosPhi_Min_NOM,			3, aData);	strcat(aData, ADR('$n'));
			strcat(aData, ADR('CosPhi_Min_TH_NOM; '));			WRITE_REAL(FDT_value.CosPhi_Min_TH_NOM,			1, aData);	strcat(aData, ADR('$n'));
			strcat(aData, ADR('CosPhi_Min_TH_s1_MAX; '));		WRITE_REAL(FDT_value.CosPhi_Min_TH_s1_MAX,		0, aData);	strcat(aData, ADR('$n'));
			strcat(aData, ADR('CosPhi_Min_TH_NOM_CNT; '));		WRITE_REAL(FDT_value.CosPhi_Min_TH_NOM_CNT,		0, aData);	strcat(aData, ADR('$n'));
			strcat(aData, ADR('CosPhi_Min_TH_s1_CNT; '));		WRITE_REAL(FDT_value.CosPhi_Min_TH_s1_CNT,		0, aData);	strcat(aData, ADR('$n'));
			strcat(aData, ADR('CosPhi_Max_NOM; '));				WRITE_REAL(FDT_value.CosPhi_Max_NOM,			3, aData);	strcat(aData, ADR('$n'));
			strcat(aData, ADR('CosPhi_Max_TH_NOM; '));			WRITE_REAL(FDT_value.CosPhi_Max_TH_NOM,			1, aData);	strcat(aData, ADR('$n'));
			strcat(aData, ADR('CosPhi_Max_TH_s1_MAX; '));		WRITE_REAL(FDT_value.CosPhi_Max_TH_s1_MAX,		0, aData);	strcat(aData, ADR('$n'));
			strcat(aData, ADR('CosPhi_Max_TH_NOM_CNT; '));		WRITE_REAL(FDT_value.CosPhi_Max_TH_NOM_CNT,		0, aData);	strcat(aData, ADR('$n'));
			strcat(aData, ADR('CosPhi_Max_TH_s1_CNT; '));		WRITE_REAL(FDT_value.CosPhi_Max_TH_s1_CNT,		0, aData);	strcat(aData, ADR('$n'));

			(* T_Main *)
			strcat(aData, ADR('T_Main_NOM; '));
			FOR iCnt:=0 TO 10 DO	WRITE_REAL(FDT_value.T_Main_NOM[iCnt],	3, aData);	END_FOR
			strcat(aData, ADR('$n'));
			strcat(aData, ADR('T_Main_TH_NOM; '));				WRITE_REAL(FDT_value.T_Main_TH_NOM,				1, aData);	strcat(aData, ADR('$n'));
			strcat(aData, ADR('T_Main_TH_s1_MAX; '));			WRITE_REAL(FDT_value.T_Main_TH_s1_MAX,			0, aData);	strcat(aData, ADR('$n'));
			strcat(aData, ADR('T_Main_TH_NOM_CNT; '));			WRITE_REAL(FDT_value.T_Main_TH_NOM_CNT,			0, aData);	strcat(aData, ADR('$n'));
			strcat(aData, ADR('T_Main_TH_s1_CNT; '));			WRITE_REAL(FDT_value.T_Main_TH_s1_CNT,			0, aData);	strcat(aData, ADR('$n'));

			(* new with V4.7 *)
			strcat(aData, ADR('Lam_Set_Min_filter_H_MAX; ')); 	WRITE_REAL(FDT_value.Lam_Set_Min_filter_H_MAX, 		3, aData);	strcat(aData, ADR('$n'));
			strcat(aData, ADR('Lam_Set_Min_filter_H_Tconst; ')); WRITE_REAL(FDT_value.Lam_Set_Min_filter_H_Tconst, 	0, aData);	strcat(aData, ADR('$n'));
			strcat(aData, ADR('Lam_Set_Max_filter_H_MAX; ')); 	WRITE_REAL(FDT_value.Lam_Set_Max_filter_H_MAX , 	3, aData);	strcat(aData, ADR('$n'));
			strcat(aData, ADR('Lam_Set_Max_filter_H_Tconst; ')); WRITE_REAL(FDT_value.Lam_Set_Max_filter_H_Tconst , 0, aData);	strcat(aData, ADR('$n'));
			strcat(aData, ADR('U_Ign_TH_MDN; ')); 				WRITE_REAL(FDT_value.U_Ign_TH_MDN , 				3, aData);	strcat(aData, ADR('$n'));
			strcat(aData, ADR('U_Ign_TH_MDN_CNT; ')); 			WRITE_REAL(FDT_value.U_Ign_TH_MDN_CNT , 			0, aData);	strcat(aData, ADR('$n'));
			strcat(aData, ADR('U_Ign_TH_s1_MAX; ')); 			WRITE_REAL(FDT_value.U_Ign_TH_s1_MAX , 				0, aData);	strcat(aData, ADR('$n'));
			strcat(aData, ADR('U_Ign_TH_s1_CNT; ')); 			WRITE_REAL(FDT_value.U_Ign_TH_s1_CNT , 				0, aData);	strcat(aData, ADR('$n'));
			strcat(aData, ADR('I_L_jumpThresh; ')); 			WRITE_REAL(FDT_value.I_L_jumpThresh , 				0, aData);	strcat(aData, ADR('$n'));
			strcat(aData, ADR('I_L_jumpTol; ')); 				WRITE_REAL(FDT_value.I_L_jumpTol , 					0, aData);	strcat(aData, ADR('$n'));
			strcat(aData, ADR('P_Act_jumpThresh; ')); 			WRITE_REAL(FDT_value.P_Act_jumpThresh , 			0, aData);	strcat(aData, ADR('$n'));
			strcat(aData, ADR('Pr_IMEP_rangeThresh; ')); 		WRITE_REAL(FDT_value.Pr_IMEP_rangeThresh , 			0, aData);	strcat(aData, ADR('$n'));
			strcat(aData, ADR('P_Set_Max_TH_SP; ')); 			WRITE_REAL(FDT_value.P_Set_Max_TH_SP , 				3, aData);	strcat(aData, ADR('$n'));
			strcat(aData, ADR('P_Set_Max_TH_SP_CNT; ')); 		WRITE_REAL(FDT_value.P_Set_Max_TH_SP_CNT , 			0, aData);	strcat(aData, ADR('$n'));
			strcat(aData, ADR('Pr_Peak_TH_MDN; ')); 			WRITE_REAL(FDT_value.Pr_Peak_TH_MDN , 				3, aData);	strcat(aData, ADR('$n'));
			strcat(aData, ADR('Pr_Peak_TH_MDN_CNT; ')); 		WRITE_REAL(FDT_value.Pr_Peak_TH_MDN_CNT , 			0, aData);	strcat(aData, ADR('$n'));
			strcat(aData, ADR('Pr_Peak2_TH_MDN; ')); 			WRITE_REAL(FDT_value.Pr_Peak2_TH_MDN , 				3, aData);	strcat(aData, ADR('$n'));
			strcat(aData, ADR('Pr_Peak2_TH_MDN_CNT; ')); 		WRITE_REAL(FDT_value.Pr_Peak2_TH_MDN_CNT , 			0, aData);	strcat(aData, ADR('$n'));
			strcat(aData, ADR('IMEP2_TH_MDN; ')); 				WRITE_REAL(FDT_value.IMEP2_TH_MDN , 				3, aData);	strcat(aData, ADR('$n'));
			strcat(aData, ADR('IMEP2_TH_MDN_CNT; ')); 			WRITE_REAL(FDT_value.IMEP2_TH_MDN_CNT , 			0, aData);	strcat(aData, ADR('$n'));
			strcat(aData, ADR('Pr_GR_Act_Max2_TH_REF; ')); 		WRITE_REAL(FDT_value.Pr_GR_Act_Max2_TH_REF , 		3, aData);	strcat(aData, ADR('$n'));
			strcat(aData, ADR('Pr_GR_Act_Max2_TH_REF_CNT; ')); 	WRITE_REAL(FDT_value.Pr_GR_Act_Max2_TH_REF_CNT , 	0, aData);	strcat(aData, ADR('$n'));
			strcat(aData, ADR('CA_PI_Duration2_TH_MDN; ')); 	WRITE_REAL(FDT_value.CA_PI_Duration2_TH_MDN , 		3, aData);	strcat(aData, ADR('$n'));
			strcat(aData, ADR('CA_PI_Duration2_TH_MDN_CNT; ')); WRITE_REAL(FDT_value.CA_PI_Duration2_TH_MDN_CNT , 	0, aData);	strcat(aData, ADR('$n'));
			strcat(aData, ADR('CA_PI_Dur_PID_Offs_TH_s1_MAX; ')); 	WRITE_REAL(FDT_value.CA_PI_Dur_PID_Offs_TH_s1_MAX , 3, aData);	strcat(aData, ADR('$n'));
			strcat(aData, ADR('CA_PI_Dur_PID_Offs_TH_s1_MAX_CNT; ')); 	WRITE_REAL(FDT_value.CA_PI_Dur_PID_Offs_TH_s1_MAX_CNT , 0, aData);	strcat(aData, ADR('$n'));
			strcat(aData, ADR('Pr_Peak_TH_LIM; ')); 			WRITE_REAL(FDT_value.Pr_Peak_TH_LIM , 				0, aData);	strcat(aData, ADR('$n'));
			strcat(aData, ADR('Pr_Peak_TH_LIM_CNT; ')); 		WRITE_REAL(FDT_value.Pr_Peak_TH_LIM_CNT , 			0, aData);	strcat(aData, ADR('$n'));
			strcat(aData, ADR('N_TCHP_A_Max_TH_REF; ')); 		WRITE_REAL(FDT_value.N_TCHP_A_Max_TH_REF , 			3, aData);	strcat(aData, ADR('$n'));
			strcat(aData, ADR('N_TCHP_A_Max_TH_REF_CNT; ')); 	WRITE_REAL(FDT_value.N_TCHP_A_Max_TH_REF_CNT , 		0, aData);	strcat(aData, ADR('$n'));
			strcat(aData, ADR('N_TCLP_A_Max_TH_REF; ')); 		WRITE_REAL(FDT_value.N_TCLP_A_Max_TH_REF , 			3, aData);	strcat(aData, ADR('$n'));
			strcat(aData, ADR('N_TCLP_A_Max_TH_REF_CNT; ')); 	WRITE_REAL(FDT_value.N_TCLP_A_Max_TH_REF_CNT , 		0, aData);	strcat(aData, ADR('$n'));

			strcat(aData, ADR('</ATD>$n'));
		END_IF
		(**** ATD- END  ****)

		strcat(aData, ADR('END OF FILE $n'));																							(* end of file *)
		iPointer	:=	save_strcat(ADR(DerString), iSize_String, iPointer, aData);														(* write line *)
		iPointer	:=	save_strcat(ADR(DerString), iSize_String, iPointer, ADR('</PBC_FILE>'));
		bWrite	:=	FALSE;																												(* buffer can start *)
		iStep	:=	_EXIST;																												(* next step *)
(** 4.8: check for existing permanent memory data module *)
	_EXIST:
			DatObjInfo_01();
			CASE  DatObjInfo_01.status OF
			_BUSY: 	iStep;
			_OKAY:	bPBC_GetFile:=	TRUE;
					iStep 		:= _WRITE;
					DatObjWrite_01.ident   	:= DatObjInfo_01.ident;
					DatObjWrite_01.len		:= pm_len;
			_DONF:	iStep		:=	_CREATE;
			ELSE	iErrorStep	:=	iStep;
					iStep		:=	_ERROR;
					iError		:=	DatObjInfo_01.status;
			END_CASE
(** 4.10: create permanent memory data module *)
	_CREATE:
		DatObjCreate_01();             			(* repeat until generation of permanent memory data module is ready *)
		CASE  DatObjCreate_01.status OF
		_BUSY:	iStep;
		_OKAY:	DatObjWrite_01.ident   	:= DatObjCreate_01.ident;		(* set identifier of permanent memory data module     	*)
				DatObjWrite_01.len		:= pm_len;
				iStep		:=	_WRITE;
		ELSE	iErrorStep	:=	iStep;
				iStep		:=	_ERROR;
				iError		:=	DatObjCreate_01.status;
		END_CASE
(** 4.10: write permanent memory data module *)
	_WRITE:
		DatObjWrite_01();
	 	CASE DatObjWrite_01.status OF
		_BUSY:	iStep;	(*mach nix*)
    	_OKAY:	iStep		:=	_HMI;
				iECB_HMI	:=	0;
				bPBC_GetFile:=	TRUE;
		ELSE	iErrorStep	:=	iStep;
				iStep		:=	_ERROR;
				iError		:=	DatObjWrite_01.status;
		END_CASE
(** 4.11.: waiting for HMI to pickup file, unlock 'DerString' *)
	_HMI:
		bECB_Lock		:=	FALSE;
		iECB_HMI		:=	iECB_HMI + 100;
		MM2VIS.bECBMem_isCreated	:= TRUE;
		IF iECB_HMI >= TIME_TO_UDINT(tiHMI_Delay) OR VIS2MM.bECBMem_isRead THEN
			iStep		:=	_DONE;
			MM2VIS.bECBMem_isCreated	:= FALSE;
			VIS2MM.bECBMem_isRead		:= FALSE;
		END_IF
(** 4.12: done *)
	_DONE:	iStep		:=	_IDLE;

(** 4.13: idle, waiting for triggers *)
	_IDLE:	iZeile		:=	0;
			iErrorStep	:=	0;
			iError		:=	0;
(** 4.14: error, waiting for cold start *)
	_ERROR:	iStep;
			bECB_Lock	:=	FALSE;

	END_CASE

(** 5: HMI Links *)

	MM2VIS.ECB.bSave	:=	iStep <> _IDLE;
	MM2VIS.ECB.bBuff	:=	bPBC_Record;
	MM2VIS.ECB.bLock	:=	iStep <> _IDLE OR bPBC_Write;
	IF bPBC_Write AND bPBC_Record AND iStep = _IDLE THEN
		MM2VIS.ECB.iStep	:=	_WAIT;
	ELSE
		MM2VIS.ECB.iStep	:=	iStep;
	END_IF

	IF tiHMI_Delay <> T#0s THEN
		rHMI_Delay	:=	LIMIT(0.0, UDINT_TO_REAL(iECB_HMI) / TIME_TO_REAL(tiHMI_Delay), 1.0);
	ELSE
		rHMI_Delay	:=	0;
	END_IF

	IF iStep = _DONE THEN
		MM2VIS.ECB.rSave	:=	1.0;
	ELSIF iStep <> _HMI THEN
		MM2VIS.ECB.rSave	:=	0.5 * INT_TO_REAL(iZeile)/INT_TO_REAL(iBufferSize);
	ELSIF iStep = _HMI THEN
		MM2VIS.ECB.rSave	:=	0.5 + 0.5 * rHMI_Delay;
	END_IF

	MM2VIS.ECB.bWarn	:=	iTC_Max = INT_TO_UINT(Buffer.iCnt_ui16_H) OR
							iEC_Max = INT_TO_UINT(Buffer.iCnt_ui16) OR
							iSC_Max = INT_TO_UINT(Buffer.iCnt_ui16_low) OR
							iPC_Max = INT_TO_UINT(Buffer.iCnt_pattern);

END_PROGRAM
```

#### PBC_Obj.var - Local variables
```iecst
(********************************************************************
 * COPYRIGHT -- INNIO Company
 ********************************************************************
 * Program: PBC_MFile
 * File: PBC_MFile.var
 * Author: 502293141
 * Created: October 23, 2014
 ********************************************************************
 * Local variables of program PBC_MFile
 ********************************************************************)
VAR
	aData : UDINT;
	aH : UDINT;
	aT : UDINT;
	strFile : STRING[50];
	ModulName : STRING[32];
	szHeader : STRING[30000];
	szData : STRING[30000];
	szTemp : STRING[10];
	strVersion : STRING[30];
	i : USINT;
	iZeile : INT;
	iIdx : INT;
	iIdx10 : INT;
	iCyl : USINT;
	bWrite : BOOL;
	iIdx1 : INT;
	iCnt : INT;
	iCnt_B : UINT;
	pm_len : UDINT := 0;
	iStep : USINT := 0;
	DatObjWrite_01 : DatObjWrite;
	DatObjInfo_01 : DatObjInfo;
	DatObjCreate_01 : DatObjCreate;
	iPointer : UDINT;
	iSize_String : UDINT;
	iCnt2 : INT;
	bTest_Ena : BOOL := 0;
	bName : BOOL := 0;
	iECB_HMI : UDINT := 0;
	rHMI_Delay : REAL;
	bPBC_GetFile : BOOL := 0;
	iAccel : INT;
	iError : UINT;
	iErrorStep : INT;
	TON_15min : TON;
	iLogicSize_1 : INT;
	iLogicSize_2 : INT;
	bSCD_Ena : BOOL := 0;
	strTemp : STRING[10];
	tiMax : TIME;
	tiMin : TIME;
	bFilled : BOOL;
END_VAR
```

### Program Logical/CBM/PBCMemV2/TCB_Buffer (IEC) - + collects data every 10ms

- TCB_Buffer.st (not readable text: treated as protected, skipped)

#### TCB_Buffer.var - Local variables
```iecst
(********************************************************************
 * COPYRIGHT -- INNIO Company
 ********************************************************************
 * Program: TCB_Buffer
 * File: TCB_Buffer.var
 * Author: 502423184
 * Created: January 18, 2018
 ********************************************************************
 * Local variables of program TCB_Buffer
 ********************************************************************)
VAR
	GetTCB_H : TCB_Header;
	GetTCB : ARRAY[0..iTCB_Max] OF TCB_In;
	iC : TCB_Cnt;
	i : UINT;
	Trace : ARRAY[0..9] OF _Tracer;
	uiTemp : UINT := 0;
	iTemp : INT := 0;
	xR_TRIG : ARRAY[0..9] OF R_TRIG := [10(0)];
	xTCB_DOW : DatObjWrite;
	xTCB_DOC : DatObjCreate;
	xTCB_DOI : DatObjInfo;
	ModulName : STRING[32];
	bTemp : BOOL := 0;
	iAvail : INT;
	iUsed : INT;
	rYourRealInputVariable : REAL;
	bCust_Trig : BOOL := 0;
	aH : UDINT;
	Z : USINT;
	rCnt_OpH : REAL;
	rCnt_Starts : REAL;
	iTCB_Status : USINT := 0;
	iTCB_Trigger : USINT;
	iCnt_Remain : INT;
	bTCB_Header : BOOL := 0;
	strFile : STRING[50];
	strTemp : STRING[10];
	iClr1 : INT := 0;
	iClr2 : INT := 0;
	iTCB_ErrorStep : USINT;
	iTCB_Error : UINT;
	iTCB_HMI : UDINT;
	iPointer : UDINT := 0;
	iStrSize : UDINT := 0;
	strData : STRING[30000];
	iIdx : UINT;
	iIdx1 : UINT;
	iTCB_Trigger_Old : USINT;
	szData : STRING[5000];
	aData : UDINT;
	iCnt : UINT;
	iCyl : USINT;
	iLine : UINT;
	strVersion : STRING[30];
	rHMI_Delay : REAL;
	rCnt_Remain : REAL;
	iCnt_10ms : INT := 0; (*TCB Ring Buffer Counter*)
	bTCB_Buffering_Ena : BOOL := FALSE; (*TCB Buffering enabled*)
	tiMax : TIME;
	tiMin : TIME;
	bFilled : BOOL;
END_VAR
```

- TCB_Functions.st (not readable text: treated as protected, skipped)

#### TCB_Functions.fun
```iecst
FUNCTION_BLOCK TCB_In
	VAR_INPUT
		rI : REAL; (*Input*)
		iI : UDINT; (*Input*)
		N : STRING[NameSize]; (*Name max 21 Characters*)
		F : USINT; (*Determines storage*)
		U : STRING[UnitSize]; (*Unit max 5 Characters*)
		C : REAL; (*Conversion factor 1 = no conversion*)
	END_VAR
	VAR_OUTPUT
		O : REAL; (*Out*)
	END_VAR
END_FUNCTION_BLOCK

FUNCTION_BLOCK TCB_Cnt
	VAR_INPUT
		E : BOOL; (*Counter ++*)
		bDEL : BOOL; (*Reset*)
		iMAX : UINT;
	END_VAR
	VAR_OUTPUT
		O : UINT; (*Out*)
		V : INT; (*Variables*)
	END_VAR
END_FUNCTION_BLOCK

FUNCTION_BLOCK TCB_Header
	VAR_INPUT
		aI : UDINT;	(* Address Real Array Input *)
		H : UDINT;	(* Header Address *)
		L : USINT;	(* Real Array Input length *)
		P : USINT;	(* Precision *)
		E : BOOL;	(* Exist *)
		N : STRING[NameSize]; (*Name max 21 Characters*)
		U : STRING[UnitSize]; (*Unit max 5 Characters*)
	END_VAR
	VAR
		iCnt : USINT;
		temp : ARRAY[0..24] OF REAL;
	END_VAR
END_FUNCTION_BLOCK
```

#### TCB_Buffer.typ - Local data types
```iecst
(********************************************************************
 * COPYRIGHT -- INNIO Company
 ********************************************************************
 * Program: TCB_Buffer
 * File: TCB_Buffer.typ
 * Author: 502423184
 * Created: January 29, 2018
 ********************************************************************
 * Local data types of program TCB_Buffer
 ********************************************************************)

TYPE
	_TracerIn : 	STRUCT
		Name : STRING[21];
		Unit : STRING[6];
		Format : USINT;
		Convert : REAL;
		Adress : STRING[100];
		Typdef : USINT;
		Record : BOOL;
	END_STRUCT;
	_TracerOut : 	STRUCT
		Adress : UDINT;
		Length : UDINT;
		rValue : REAL;
	END_STRUCT;
	_Tracer : 	STRUCT
		In : _TracerIn;
		Out : _TracerOut;
	END_STRUCT;
END_TYPE
```

### Package Logical/CBM/Statistic - Start Up Statistic

### Statistic.var - Package variables
```iecst
(********************************************************************
 * COPYRIGHT -- INNIO Company
 ********************************************************************
 * Package: Statistic
 * File: Statistic.var
 * Author: 502423184
 * Created: May 18, 2015
 ********************************************************************
 * Variables of package Statistic
 ********************************************************************)
VAR
	bStat_Trigger : BOOL := FALSE;
	Stat : _StatBuffer; (*circular buffer*)
	bStat_Sync_Max : BOOL;
	rP_Sync_Max : REAL;
	rI_Sync_L1_Max : REAL;
	rI_Sync_L2_Max : REAL;
	rI_Sync_L3_Max : REAL;
	bStat_OS_Max : BOOL;
	rP_OS_Max : REAL;
	rP_Set_OS_Max : REAL;
	Err : _ErrStat;
	ErrName : ARRAY[0..20] OF _NameErr := [21(0)];
END_VAR
```

### Statistic.typ - Package data types
```iecst
(********************************************************************
 * COPYRIGHT -- INNIO Company
 ********************************************************************
 * Package: Statistic
 * File: Statistic.typ
 * Author: 502423184
 * Created: May 18, 2015
 ********************************************************************
 * Data types of package Statistic
 ********************************************************************)

TYPE
	_pmCBM : 	STRUCT
		Stat : _StatBuffer;
		Err : _ErrStat;
	END_STRUCT;
	_ErrStat : 	STRUCT
		tTS_Reset : tTimeStamp_typ;
		Size : UINT;
		iCnt_OH_Reset : DINT;
		xErr : ARRAY[0..ErrCntSize]OF ErrCnt_FUB;
	END_STRUCT;
	_StrData : 	STRUCT
		str : STRING[30];
	END_STRUCT;
	_StringData : 	STRUCT
		Name : STRING[NameSize];
		Data : ARRAY[0..StatSize]OF _StrData;
		Skip : BOOL;
	END_STRUCT;
	_BoolData : 	STRUCT
		Name : STRING[NameSize];
		Data : ARRAY[0..StatSize]OF BOOL;
		Skip : BOOL;
	END_STRUCT;
	_UsintData : 	STRUCT
		Name : STRING[NameSize];
		Unit : STRING[UnitSize];
		Data : ARRAY[0..StatSize]OF USINT;
		Skip : BOOL;
	END_STRUCT;
	_RealData : 	STRUCT
		Name : STRING[NameSize];
		Unit : STRING[UnitSize];
		Deci : USINT;
		Data : ARRAY[0..StatSize]OF REAL;
		Skip : BOOL;
	END_STRUCT;
	_NameErr : 	STRUCT
		str : STRING[21];
	END_STRUCT;
	_StatBuffer : 	STRUCT
		r : ARRAY[0..StatRealSize]OF _RealData; (*real data*)
		rSize : USINT;
		b : ARRAY[0..StatBoolSize]OF _BoolData; (*boolean data*)
		bSize : USINT;
		i : ARRAY[0..StatIntSize]OF _UsintData; (*unsigned short integer data*)
		iSize : USINT;
		s : ARRAY[0..StatStrSize]OF _StringData; (*String data*)
		sSize : USINT;
		iIdx : USINT; (*current data Index*)
		bFilled : BOOL; (*is buffer filled?*)
	END_STRUCT;
END_TYPE
```

### Program Logical/CBM/Statistic/Stat100ms (IEC, version 4.14.0) - + Statistic package

- Stat100msCyclic.st (not readable text: treated as protected, skipped)

- Stat100msInit.st (not readable text: treated as protected, skipped)

#### Stat100ms.var - Local variables
```iecst
VAR
	xTON_WritePMEM : TON;
	write_once : BOOL;
	pmCBM : _pmCBM;
	ulChecksum : UDINT;
	ulPMPointer : UDINT;
	pm_len : UDINT;
	ulChkValue : UDINT;
	ulChecksumOld : UDINT;
	bWriteDataObj : BOOL;
	DatObjWrite_01 : DatObjWrite;
	pmPrstWriteCnt : UINT;
	pm_Error : UINT;
	bErrPermSlowDown : BOOL;
	xTON_WarnDelay : TON;
	ModulName : STRING[32];
	DatObjInfo_01 : DatObjInfo;
	pm_id : UDINT;
	pm_p : UDINT;
	bCreateDataObj : BOOL;
	perm_vers : UINT;
	DatObjRead_01 : DatObjRead;
	DatObjDelete_PermMem : DatObjDelete;
	DatObjCreate_01 : DatObjCreate;
	rP_Targ : REAL;
	rP_Targ_old : REAL;
	xTON_Nox : TON;
	bNox : BOOL; (*bit if Nox time recording is already done*)
	xTON_Set : TON;
	bSet : BOOL; (*bit if Settling time recording is already done*)
	rPr_NOx_Lim : REAL;
	iStat_State : INT;
	xTP_MaxCurr : TP;
	xTP_PelMax : TP;
	xTP_MSSTA : TP;
	k : INT;
	i : INT;
	szAlarm : STRING[6];
	j : USINT;
	m : INT;
	rPr_Starter : ARRAY[0..49] OF REAL;
	bAlarm_Ena : BOOL;
	bNoxGoUp : BOOL;
	xTON_NoxGoUp : TON;
	ERR_NOERROR : UINT := 0;
	bSection : ARRAY[0..5] OF BOOL;
	tiSection : ARRAY[0..5] OF TIME;
	ii : USINT;
	iCnt_AllStarts : USINT;
	iCnt_ManAbort : USINT;
	iCnt_Success : USINT;
	iCnt_SuccessReli : USINT;
	bSuccess : ARRAY[0..StatSize] OF BOOL;
	rStartReli : REAL;
	iCnt_End : USINT;
	rTi_Prep : ARRAY[0..2] OF REAL;
	rTi_Speedup : ARRAY[0..2] OF REAL;
	rTi_Load : ARRAY[0..2] OF REAL;
	iCnt_GoodData : USINT;
	iCnt_Begin : USINT;
	bOverFlow : BOOL;
	bBreak : BOOL;
	iCnt_Begin10 : USINT;
	iCnt_Found10 : USINT;
	rTi_Start : ARRAY[0..2] OF REAL;
	rTi_Sync : ARRAY[0..2] OF REAL;
	iCnt : USINT;
	iCnt_rpm : USINT;
	TOF_A_STRT : TOF;
	bTest_Statistic : BOOL;
	str_temp : STRING[5];
	iDays_SinceStart : INT;
	rHours_SinceStart : REAL;
	rE_SinceStart : REAL;
	rTi_SumLoad : REAL;
	rTi_SumSync : REAL;
	rTi_SumNOx : REAL;
	rTi_Stat_Max : REAL;
	xFILTER_dP : FILTER_R;
	xTON_1s : TON;
	xTON_Show_Ramp : TON;
	rP_Old_1s : REAL;
	ti_Timer : TIME;
	tiStart_PreLube : TIME;
	tiDone_PreLube : TIME;
	tiStart_Scav : TIME;
	tiDone_Scav : TIME;
	tiStart_SlowTurn : TIME;
	tiDone_SlowTurn : TIME;
	tiStart_GasLeak : TIME;
	tiDone_GasLeak : TIME;
	xTON_GCB : TON;
	bDone_PreLube : BOOL;
	bStart_PreLube : BOOL;
	bDone_GasLeak : BOOL;
	bStart_GasLeak : BOOL;
	bDone_SlowTurn : BOOL;
	bStart_SlowTurn : BOOL;
	bDone_Scav : BOOL;
	bStart_Scav : BOOL;
	bSync : BOOL := 0;
	ti_Conrod : TIME;
	tiFiring : ARRAY[0..49] OF TIME;
	rN_Firing : ARRAY[0..49] OF REAL;
	bStart_StartDur : BOOL := 0;
	bDone_StartDur : BOOL := 0;
	rN_StarterSum : ARRAY[0..49] OF REAL;
	rN_Starter_Sum : REAL;
	tiStart_StartDur : TIME := 0;
	rN_Anz : REAL;
	bTurbo_Hot : BOOL := 0;
	bSet_EngRuns : BOOL := 0;
	rN_Oil : REAL;
	rAll : REAL;
	rT_MB_Max : REAL;
	iNum_MBT_Max : USINT;
	iCnt_Hot : USINT;
	iCnt_Warm : USINT;
	iCnt_Cold : USINT;
	iCnt_Unknown : USINT;
	rTi_Starter : ARRAY[0..2] OF REAL;
	rN_Starter : ARRAY[0..2] OF REAL;
	xGetTime : DTGetTime := (0);
	DT_EngStop : DATE_AND_TIME;
	rN_Buffer : ARRAY[0..24] OF REAL;
	iCnt_Buf : USINT;
	rN_Dot_Dot : ARRAY[0..49] OF REAL;
	rN_Dot : REAL;
	rN_Dot_Old : REAL;
	rN_Avg : REAL;
	rN_Avg_Old : REAL;
	iPos_N_Dot_Dot_Max : USINT;
	iLastRunInfo : USINT;
	bSkipData : BOOL := 0;
	ti_Sync_Dur : TIME;
	tiPurge_Dur : TIME;
	tiWait4StartTempRel : TIME;
END_VAR
VAR CONSTANT
	_HOT : USINT := 3;
	_WARM : USINT := 2;
	_COLD : USINT := 1;
	_ALLRIGHT : INT := 0;
	_ENG_FAIL : INT := -1;
	_MAN_FAIL : INT := -2;
	_P_SET_FAIL : INT := -3;
END_VAR
VAR
	bSec3_Hold : BOOL := 0;
	rN_Dot_Dot_Max : REAL;
END_VAR
```

#### Stat100msData.var - Local variables
```iecst
VAR
	Year : USINT;
	Month : USINT;
	Day : USINT;
	Hour : USINT;
	Minute : USINT;
	Cyl_EGT_Max : USINT;
	Cyl_CBT_Max : USINT;
	Num_MBT_Max : USINT;
	ContGen : USINT;
	TripSec : USINT;
	TripPrio : USINT;
	WaterLeak : USINT;
	FastStart : USINT;
	TripID : USINT;
	Ti_Set : USINT;
	Ti_Prep : USINT;
	Ti_Speedup : USINT;
	Ti_Sync : USINT;
	Ti_Load : USINT;
	Ti_Start : USINT;
	Ti_Starter : USINT;
	Ti_Str_n100 : USINT;
	Ti_NOx : USINT;
	P_Set_MaxOS : USINT;
	P_MaxOS : USINT;
	P_Nom : USINT;
	P_Targ : USINT;
	P_Sync_Max : USINT;
	P_RampSet : USINT;
	T_Oil2 : USINT;
	T_Oil4 : USINT;
	T_Oil75 : USINT;
	T_Wat2 : USINT;
	T_Wat4 : USINT;
	T_Wat75 : USINT;
	T_T3LP_A : USINT;
	T_T3LP_B : USINT;
	T_T3HP_A : USINT;
	T_T3HP_B : USINT;
	T_EG_Max : USINT;
	T_CB_Max : USINT;
	T_MB_Max : USINT;
	I_Sync_L1 : USINT;
	I_Sync_L2 : USINT;
	I_Sync_L3 : USINT;
	Pr_Starter : USINT;
	Pr_Vessel : USINT;
	Pr_GR_n100 : USINT;
	Pr_GR_n200 : USINT;
	Pr_GR_n500 : USINT;
	Pr_GR_n890 : USINT;
	Pr_PC_n100 : USINT;
	Pr_PC_n200 : USINT;
	Pr_PC_n500 : USINT;
	Pr_PC_n890 : USINT;
	MFB50 : USINT;
	T_AirIn : USINT;
	T_T2s2 : USINT;
	T_T2s4 : USINT;
	T_T2s75 : USINT;
	Starts : USINT;
	OpHours : USINT;
	CQMax : ARRAY[0..24] OF USINT;
	Ti_PreLube : USINT;
	Ti_GasLeak : USINT;
	Ti_SlowTurn : USINT;
	Ti_Scav : USINT;
	Ti_CR_OutIn : ARRAY[0..24] OF USINT;
	Ti_CR_Out : ARRAY[0..24] OF USINT;
	Ti_CR_In : ARRAY[0..24] OF USINT;
	Ti_Firing : USINT;
	N_Firing : USINT;
	T_EG_Sync_Max : USINT;
	T_EG_Sync_Med : USINT;
	EngTemp : USINT;
	N_Starter : USINT;
	Ti_StartDur : USINT;
	Ti_LastRun : USINT;
	F_DiffMax : USINT;
	F_DiffMin : USINT;
	U_DiffMax : USINT;
	Ang_DiffMax : USINT;
	Ti_RelAux : USINT;
	LastRunInfo : USINT;
	Knck_Int_Max : USINT;
	Misf_Int_Max : USINT;
	Ti_Sync_Dur : USINT;
	CombAnomaly : USINT;
	Ti_Purge_Dur : USINT;
	Ti_Wait4StartTempRel : USINT;
END_VAR
```

### Program Logical/CBM/Statistic/Stat10ms (IEC, version 4.06.1) - + Part of statistic package

- Stat10ms.st (not readable text: treated as protected, skipped)

### Program Logical/CBM/Statistic/Stat_Obj (IEC, version 4.14.0) - Save Files
